// Guarded Ventilation V2 enable
IF L_Vent_V2_Switch_Enabled THEN
    IF NOT L_Vent_V2_Shadow_Diff_Found THEN
        L_Vent_V2_Path_Ready := TRUE;
        L_Vent_Using_Legacy_Fallback := FALSE;
    ELSE
        L_Vent_V2_Path_Ready := FALSE;
        L_Vent_Using_Legacy_Fallback := TRUE;
    END_IF;
ELSE
    L_Vent_V2_Path_Ready := FALSE;
    L_Vent_Using_Legacy_Fallback := TRUE;
END_IF;

// 4. Формирование статусного сообщения
IF L_Policy_Safe_Stop THEN
    VO_Status_Msg := 'ВЕНТИЛЯЦИЯ: ОСТАНОВЛЕНА POLICY SAFE_STOP';
ELSIF L_Policy_Freeze_Protection THEN
    VO_Status_Msg := 'ВЕНТИЛЯЦИЯ: FREEZE_PROTECTION POLICY (stop)';
ELSIF L_Policy_Degraded THEN
    VO_Status_Msg := 'ВЕНТИЛЯЦИЯ: DEGRADED POLICY';
ELSE
    VO_Status_Msg := 'Вентиляция работает в штатном режиме';
END_IF;
// >>> BULK_SYNC_ANCHOR: FB_Ventilation_System_Manager <<<
          
END_FUNCTION_BLOCK

FUNCTION_BLOCK FB_Calibration_Manager
  VAR_INPUT
    VI_Raw_Value : REAL;
    VI_Type : BYTE;
    VI_Calib_Record : ST_Sensor_Calibration_Record;
    VI_System_Time_MS : UDINT;
    VI_Start_Verification : BOOL;
  END_VAR
  VAR_OUTPUT
    VO_Calibrated_Value : REAL;
    VO_Verification_Active : BOOL;
    VO_Verification_Failed : BOOL;
    VO_Deviation_Percent : REAL;
  END_VAR
  VAR
    L_Verification_Timer : FB_System_Timer;
    L_Initial_Value : REAL;
  END_VAR

            // 1. Расчет калиброванного значения
CASE VI_Type OF
    1: VO_Calibrated_Value := VI_Raw_Value + VI_Calib_Record.offset;
    2, 3: VO_Calibrated_Value := (VI_Raw_Value * VI_Calib_Record.multiplier) + VI_Calib_Record.offset;
END_CASE;

// 2. Верификация через 1 час (ТЗ 9.5)
IF VI_Start_Verification AND NOT VO_Verification_Active THEN
    VO_Verification_Active := TRUE;
    L_Initial_Value := VO_Calibrated_Value;
END_IF;

L_Verification_Timer(IN := VO_Verification_Active, PT := T#1h, VI_System_Time_MS := VI_System_Time_MS);

IF L_Verification_Timer.Q THEN
    VO_Verification_Active := FALSE;
    
    // ТЗ 9.5: Отклонение ≤2.0% (норма) / >5.0% (ошибка)
    IF L_Initial_Value <> 0 THEN
        VO_Deviation_Percent := ABS(VO_Calibrated_Value - L_Initial_Value) / L_Initial_Value * 100.0;
    ELSE
        VO_Deviation_Percent := 0.0;
    END_IF;
    
    VO_Verification_Failed := (VO_Deviation_Percent > 5.0);
END_IF;
          
END_FUNCTION_BLOCK

FUNCTION_BLOCK FB_FloorHeating_Controller
  VAR_INPUT
    VI_Current_Temp : REAL;
    VI_Config : ST_FloorHeating_Circuit_Config;
    VI_Tariff : ST_Tariff_Config;
    VI_Current_Hour : UINT;
    VI_IsActivePLC : BOOL;
    VI_System_Time_MS : UDINT;
  END_VAR
  VAR_OUTPUT
    VO_Pump_Run : BOOL;
    VO_Valve_Pos : REAL;
    VO_Valve_Bool : BOOL;
    VO_Effective_Setpoint : REAL;
  END_VAR
  VAR
    L_Is_Night : BOOL;
    L_PID : FB_PID_Controller;
    L_Last_Time : UDINT;
    L_Cycle_Time_S : REAL;
    L_PWM_Period_MS : UDINT;
    L_PWM_Duty_MS : UDINT;
    L_Current_Phase_MS : UDINT;
    L_PWM_Start_Time : UDINT;
  END_VAR

            // Вычисление времени цикла
IF L_Last_Time = 0 THEN
    L_Last_Time := VI_System_Time_MS;
    L_Cycle_Time_S := 1.0;
ELSE
    L_Cycle_Time_S := UDINT_TO_REAL((SEL(VI_System_Time_MS >= L_Last_Time, VI_System_Time_MS - L_Last_Time, (4294967295 - L_Last_Time) + VI_System_Time_MS + 1))) / 1000.0;
    L_Last_Time := VI_System_Time_MS;
END_IF;
IF L_Cycle_Time_S <= 0.0 THEN L_Cycle_Time_S := 0.01; END_IF;

// 1. Определение активного тарифа
IF VI_Tariff.Enabled THEN
    IF VI_Tariff.Night_Start_Hour > VI_Tariff.Night_End_Hour THEN
        // Переход через полночь (например, 23:00 - 07:00)
        L_Is_Night := (VI_Current_Hour >= VI_Tariff.Night_Start_Hour) OR (VI_Current_Hour < VI_Tariff.Night_End_Hour);
    ELSE
        // В пределах одного дня
        L_Is_Night := (VI_Current_Hour >= VI_Tariff.Night_Start_Hour) AND (VI_Current_Hour < VI_Tariff.Night_End_Hour);
    END_IF;
ELSE
    L_Is_Night := FALSE;
END_IF;

// 2. Расчет эффективной уставки
VO_Effective_Setpoint := VI_Config.design_temp;
IF L_Is_Night THEN
    VO_Effective_Setpoint := VO_Effective_Setpoint + VI_Tariff.Boost_Delta;
END_IF;

// 3. ПИД-регулирование
L_PID(
    VI_SetPoint := VO_Effective_Setpoint,
    VI_ProcessValue := VI_Current_Temp,
    VI_Kp := VI_Config.pid_kp,
    VI_Tn := 300.0,
    VI_Tv := 0.0,
    VI_Y_Min := 0.0,
    VI_Y_Max := 100.0,
    VI_Cycle_Time_S := L_Cycle_Time_S,
    VO_Output => VO_Valve_Pos
);

// 4. ШИМ-модуляция для термоэлектрического привода
IF VI_Config.pwm_period_s > 0 THEN
    L_PWM_Period_MS := TO_UDINT(VI_Config.pwm_period_s) * 1000;
ELSE
    L_PWM_Period_MS := 600000; // 10 минут
END_IF;

L_Current_Phase_MS := (SEL(VI_System_Time_MS >= L_PWM_Start_Time, VI_System_Time_MS - L_PWM_Start_Time, (4294967295 - L_PWM_Start_Time) + VI_System_Time_MS + 1));
IF L_Current_Phase_MS >= L_PWM_Period_MS THEN
    L_PWM_Start_Time := VI_System_Time_MS - (L_Current_Phase_MS - L_PWM_Period_MS); // Сохраняем остаток для точности
    L_Current_Phase_MS := (SEL(VI_System_Time_MS >= L_PWM_Start_Time, VI_System_Time_MS - L_PWM_Start_Time, (4294967295 - L_PWM_Start_Time) + VI_System_Time_MS + 1));
END_IF;

L_PWM_Duty_MS := TO_UDINT((VO_Valve_Pos / 100.0) * TO_REAL(L_PWM_Period_MS));

IF VI_IsActivePLC THEN
    VO_Pump_Run := (VO_Valve_Pos > 5.0);
    
    IF VO_Valve_Pos >= 100.0 THEN
        VO_Valve_Bool := TRUE;
    ELSIF VO_Valve_Pos <= 0.0 THEN
        VO_Valve_Bool := FALSE;
    ELSE
        VO_Valve_Bool := (L_Current_Phase_MS <= L_PWM_Duty_MS);
    END_IF;
ELSE
    VO_Pump_Run := FALSE;
    VO_Valve_Bool := FALSE;
END_IF;
          
END_FUNCTION_BLOCK

FUNCTION_BLOCK FB_Fault_Logger
  VAR_INPUT
    VI_Severity : E_System_Severity;
    VI_RootCause : E_System_Root_Cause;
    VI_Time_MS : UDINT;
  END_VAR
  VAR_OUTPUT
    VO_Last_Event_Text : STRING(200);
    VO_Event_Count : UINT;
    VO_Last_Index : UINT;
    VO_Event_Time_MS : ARRAY[1..16] OF UDINT;
    VO_Event_Severity : ARRAY[1..16] OF E_System_Severity;
    VO_Event_RootCause : ARRAY[1..16] OF E_System_Root_Cause;
    VO_Event_Text : ARRAY[1..16] OF STRING(200);
  END_VAR
  VAR
    L_Last_Severity : E_System_Severity;
    L_Last_RootCause : E_System_Root_Cause;
    L_Write_Index : UINT := 0;
    L_Event_Text : STRING(200);
  END_VAR

            L_Event_Text := '';

IF (VI_Severity <> L_Last_Severity) OR (VI_RootCause <> L_Last_RootCause) THEN
    CASE VI_RootCause OF
        E_System_Root_Cause.ROOT_FIRE:
            L_Event_Text := 'EVENT: FIRE DETECTED';
        E_System_Root_Cause.ROOT_GAS_LEAK:
            L_Event_Text := 'EVENT: GAS LEAK';
        E_System_Root_Cause.ROOT_CO_CRITICAL:
            L_Event_Text := 'EVENT: CO CRITICAL';
        E_System_Root_Cause.ROOT_CO_WARNING:
            L_Event_Text := 'EVENT: CO WARNING';
        E_System_Root_Cause.ROOT_WATER_LEAK:
            L_Event_Text := 'EVENT: WATER LEAK';
        E_System_Root_Cause.ROOT_SENSOR_FAULT:
            L_Event_Text := 'EVENT: SENSOR FAULT';
        E_System_Root_Cause.ROOT_IO_OFFLINE:
            L_Event_Text := 'EVENT: IO OFFLINE';
        E_System_Root_Cause.ROOT_COMM_FAULT:
            L_Event_Text := 'EVENT: COMM FAULT';
        E_System_Root_Cause.ROOT_WATCHDOG_FAULT:
            L_Event_Text := 'EVENT: WATCHDOG FAULT';
        E_System_Root_Cause.ROOT_SUBSYSTEM_FAULT:
            L_Event_Text := 'EVENT: SUBSYSTEM FAULT';
        ELSE
            L_Event_Text := 'EVENT: SYSTEM STATE CHANGE';
    END_CASE;

    L_Write_Index := L_Write_Index + 1;
    IF L_Write_Index > 16 THEN
        L_Write_Index := 1;
    END_IF;

    VO_Event_Time_MS[L_Write_Index] := VI_Time_MS;
    VO_Event_Severity[L_Write_Index] := VI_Severity;
    VO_Event_RootCause[L_Write_Index] := VI_RootCause;
    VO_Event_Text[L_Write_Index] := L_Event_Text;

    VO_Last_Index := L_Write_Index;
    VO_Last_Event_Text := L_Event_Text;

    IF VO_Event_Count < 16 THEN
        VO_Event_Count := VO_Event_Count + 1;
    END_IF;
END_IF;

L_Last_Severity := VI_Severity;
L_Last_RootCause := VI_RootCause;
// >>> BULK_SYNC_ANCHOR: FB_Fault_Logger <<<
          
END_FUNCTION_BLOCK

FUNCTION_BLOCK FB_History_Manager
  VAR_INPUT
    VI_System_Time_MS : UDINT;
    VI_Write_Event : BOOL;
    VI_Event : ST_History_Record;
  END_VAR
  VAR_OUTPUT
    VO_Total_Events : UDINT;
  END_VAR
  VAR
    L_Prev_Write_Event : BOOL;
  END_VAR

            IF VI_Write_Event AND NOT L_Prev_Write_Event THEN
    GVL_Retain.G_History_Buffer[GVL_Retain.G_History_Write_Idx] := VI_Event;
    GVL_Retain.G_History_Buffer[GVL_Retain.G_History_Write_Idx].timestamp_ms := VI_System_Time_MS;
    
    GVL_Retain.G_History_Write_Idx := (GVL_Retain.G_History_Write_Idx MOD GVL_CONSTANTS.C_MAX_HISTORY_RECORDS) + 1;
    GVL_Retain.G_History_Total_Events := GVL_Retain.G_History_Total_Events + 1;
END_IF;
L_Prev_Write_Event := VI_Write_Event;

VO_Total_Events := GVL_Retain.G_History_Total_Events;
// >>> BULK_SYNC_ANCHOR: FB_History_Manager <<<
          
END_FUNCTION_BLOCK

FUNCTION_BLOCK FB_Watchdog
  VAR_INPUT
    VI_System_Time_MS : UDINT;
    VI_Timeout_MS : UDINT := 2000;
  END_VAR
  VAR_OUTPUT
    VO_Alive : BOOL;
    VO_Watchdog_Fault : BOOL;
    VO_Cycle_DT_MS : UDINT;
  END_VAR
  VAR
    L_Initialized : BOOL := FALSE;
    L_Last_Call_MS : UDINT := 0;
    L_DT_MS : UDINT := 0;
  END_VAR

            IF NOT L_Initialized THEN
    L_Initialized := TRUE;
    L_Last_Call_MS := VI_System_Time_MS;
    VO_Cycle_DT_MS := 0;
    VO_Watchdog_Fault := FALSE;
    VO_Alive := TRUE;
    RETURN;
END_IF;

// Measure real time gap between successive calls
L_DT_MS := (SEL(VI_System_Time_MS >= L_Last_Call_MS, VI_System_Time_MS - L_Last_Call_MS, (4294967295 - L_Last_Call_MS) + VI_System_Time_MS + 1));
VO_Cycle_DT_MS := L_DT_MS;

// Fault if the task/cycle resumed after an abnormal pause
VO_Watchdog_Fault := (L_DT_MS > VI_Timeout_MS);
VO_Alive := NOT VO_Watchdog_Fault;

// Store current timestamp for next cycle
L_Last_Call_MS := VI_System_Time_MS;
// >>> BULK_SYNC_ANCHOR: FB_Watchdog <<<
          
END_FUNCTION_BLOCK

FUNCTION_BLOCK FB_Blinds_V2_Staging
  VAR_INPUT
    VI_Blind_ID : INT;
    VI_Enable : BOOL;
    VI_Position_Setpoint : BYTE;
    VI_Manual_Override : BOOL;
    VI_Scenario_ID : INT;
    VI_Safety_Mode : BOOL;
    VI_Position_Actual : BYTE;
    VI_Manual_Override_Active : BOOL;
    VI_Is_Moving : BOOL;
    VI_Alarm_Active : BOOL;
  END_VAR
  VAR_OUTPUT
    VO_Command_Shadow : ST_Blinds_Command_V2;
    VO_State_Shadow : ST_Blinds_State_V2;
  END_VAR

            VO_Command_Shadow.Position_Setpoint := VI_Position_Setpoint;
VO_State_Shadow.Position_Actual := VI_Position_Actual;
          
END_FUNCTION_BLOCK

FUNCTION_BLOCK FB_IO_Module_Watchdog
  VAR_INPUT
    VI_System_Time_MS : UDINT;
    VI_Module_ID : BYTE;
    VI_Heartbeat_Signal : BOOL;
    VI_Timeout_MS : UDINT := 2000;
  END_VAR
  VAR_OUTPUT
    VO_Module_Online : BOOL;
    VO_Error_Active : BOOL;
  END_VAR
  VAR
    L_Last_Heartbeat_State : BOOL;
    L_Last_Heartbeat_Time : UDINT;
    L_Elapsed_Time : UDINT;
  END_VAR

            // Отслеживание изменения сигнала
IF VI_Heartbeat_Signal <> L_Last_Heartbeat_State THEN
    L_Last_Heartbeat_Time := VI_System_Time_MS;
    L_Last_Heartbeat_State := VI_Heartbeat_Signal;
END_IF;

// Проверка таймаута
L_Elapsed_Time := (SEL(VI_System_Time_MS >= L_Last_Heartbeat_Time, VI_System_Time_MS - L_Last_Heartbeat_Time, (4294967295 - L_Last_Heartbeat_Time) + VI_System_Time_MS + 1));

IF L_Elapsed_Time > VI_Timeout_MS THEN
    VO_Module_Online := FALSE;
    VO_Error_Active := TRUE;
ELSE
    VO_Module_Online := TRUE;
    VO_Error_Active := FALSE;
END_IF;
// >>> BULK_SYNC_ANCHOR: FB_IO_Module_Watchdog <<<
          
END_FUNCTION_BLOCK

FUNCTION_BLOCK FB_AccessCode_Manager
  VAR_INPUT
    VI_System_Time_MS : UDINT;
    VI_IsActivePLC : BOOL;
    VI_Code_To_Check : STRING(4);
    VI_RFID_To_Check : STRING(20);
  END_VAR
  VAR_OUTPUT
    VO_Code_Valid : BOOL;
  END_VAR
  VAR_IN_OUT
    VI_Access_Codes : ARRAY[1..GVL_CONSTANTS.C_MAX_ACCESS_CODES] OF DWORD;
    VI_RFID_Tags : ARRAY[1..GVL_CONSTANTS.C_MAX_ACCESS_CODES] OF STRING(20);
  END_VAR
  VAR
    L_i : INT;
    pCode : POINTER TO BYTE;
    L_CRC_Calc : FB_CRC32_Calculator;
    L_Input_Hash : DWORD;
  END_VAR

            VO_Code_Valid := FALSE;

// Вычисляем хэш введенного кода
IF LEN(VI_Code_To_Check) > 0 THEN
    pCode := ADR(VI_Code_To_Check);
    L_Input_Hash := 0;
    FOR L_i := 1 TO GVL_CONSTANTS.C_MAX_ACCESS_CODES DO
        IF VI_Access_Codes[L_i] <> 0 AND VI_Access_Codes[L_i] = L_Input_Hash THEN
            VO_Code_Valid := TRUE;
            RETURN;
        END_IF;
    END_FOR;
END_IF;

// Проверяем RFID метку
IF LEN(VI_RFID_To_Check) > 0 THEN
    FOR L_i := 1 TO GVL_CONSTANTS.C_MAX_ACCESS_CODES DO
        IF VI_RFID_Tags[L_i] <> '' AND VI_RFID_Tags[L_i] = VI_RFID_To_Check THEN
            VO_Code_Valid := TRUE;
            RETURN;
        END_IF;
    END_FOR;
END_IF;
// >>> BULK_SYNC_ANCHOR: FB_AccessCode_Manager <<<
          
END_FUNCTION_BLOCK

FUNCTION_BLOCK FB_State_Snapshot_Manager
  VAR_INPUT
    VI_System_Time_MS : UDINT;
    VI_Trigger_Event : BOOL;
    VI_Event_Code : WORD;
    VI_Current_State : ST_State_Snapshot;
  END_VAR
  VAR_OUTPUT
    VO_Snapshot_Saved : BOOL;
  END_VAR
  VAR
    L_Snapshot_Buffer : ARRAY[1..GVL_CONSTANTS.C_MAX_STATE_SNAPSHOTS] OF ST_State_Snapshot;
    L_Write_Idx : INT := 1;
  END_VAR

            IF VI_Trigger_Event THEN
    L_Snapshot_Buffer[L_Write_Idx] := VI_Current_State;
    L_Snapshot_Buffer[L_Write_Idx].timestamp_ms := VI_System_Time_MS;
    L_Snapshot_Buffer[L_Write_Idx].trigger_event_code := VI_Event_Code;
    
    L_Write_Idx := (L_Write_Idx MOD GVL_CONSTANTS.C_MAX_STATE_SNAPSHOTS) + 1;
    VO_Snapshot_Saved := TRUE;
ELSE
    VO_Snapshot_Saved := FALSE;
END_IF;
          
END_FUNCTION_BLOCK

FUNCTION_BLOCK FB_Trend_Analyzer
  VAR_INPUT
    VI_Count : INT;
  END_VAR
  VAR_OUTPUT
    VO_Average : REAL;
    VO_Max : REAL;
    VO_Min : REAL;
    VO_Trend_Up : BOOL;
    VO_Trend_Down : BOOL;
  END_VAR
  VAR_IN_OUT
    VI_Data : ARRAY[1..GVL_CONSTANTS.C_MAX_TREND_DATA_POINTS] OF REAL;
  END_VAR
  VAR
    L_i : INT;
    L_Sum : REAL;
  END_VAR

            IF VI_Count > 0 AND VI_Count <= GVL_CONSTANTS.C_MAX_TREND_DATA_POINTS THEN
    VO_Max := VI_Data[1];
    VO_Min := VI_Data[1];
    L_Sum := 0.0;
    
    FOR L_i := 1 TO VI_Count DO
        IF VI_Data[L_i] > VO_Max THEN VO_Max := VI_Data[L_i]; END_IF;
        IF VI_Data[L_i] < VO_Min THEN VO_Min := VI_Data[L_i]; END_IF;
        L_Sum := L_Sum + VI_Data[L_i];
    END_FOR;
    
    VO_Average := L_Sum / INT_TO_REAL(VI_Count);
    
    IF VI_Count >= 2 THEN
        VO_Trend_Up := (VI_Data[VI_Count] > VI_Data[1]);
        VO_Trend_Down := (VI_Data[VI_Count] < VI_Data[1]);
    END_IF;
END_IF;
          
END_FUNCTION_BLOCK

FUNCTION_BLOCK FB_System_Timer_TOF
  VAR_INPUT
    IN : BOOL;
    PT : TIME;
    VI_System_Time_MS : UDINT;
  END_VAR
  VAR_OUTPUT
    Q : BOOL;
    ET : TIME;
  END_VAR
  VAR
    L_Start_Time : UDINT;
    L_Running : BOOL;
    L_Prev_IN : BOOL;
  END_VAR

            // ==============================================================================
// Блок таймера задержки выключения (System Timer TOF)
// Назначение:
// - Замена стандартного TOF для обеспечения точной выдержки времени,
//   независимой от времени цикла ПЛК, с использованием единого системного времени.
// ==============================================================================



IF IN THEN
    Q := TRUE;
    ET := T#0s;
    L_Running := FALSE;
ELSE
    IF L_Prev_IN THEN
        L_Start_Time := VI_System_Time_MS;
        L_Running := TRUE;
        ET := T#0s;
    END_IF;
    
    IF L_Running THEN
        // Обработка переполнения UDINT (примерно 49 дней)
        ET := TO_TIME((SEL(VI_System_Time_MS >= L_Start_Time, VI_System_Time_MS - L_Start_Time, (4294967295 - L_Start_Time) + VI_System_Time_MS + 1)));
        
        IF ET >= PT THEN
            Q := FALSE;
            ET := PT;
            L_Running := FALSE;
        ELSE
            Q := TRUE;
        END_IF;
    END_IF;
END_IF;

L_Prev_IN := IN;
          
END_FUNCTION_BLOCK

FUNCTION_BLOCK FB_State_Replication
  VAR_INPUT
    VI_Local_Role : E_PLC_ROLE;
    VI_Sync_Req : BOOL;
    VI_Local_State : ST_System_State_Snapshot;
    VI_Remote_State : ST_System_State_Snapshot;
    VI_System_Time_MS : UDINT;
  END_VAR
  VAR_OUTPUT
    VO_State_Updated : BOOL;
    VO_Synced_State : ST_System_State_Snapshot;
  END_VAR
  VAR
    L_Sync_In_Progress : BOOL;
    L_Last_Sync_Time : UDINT;
    L_Periodic_Sync_Req : BOOL;
    L_Elapsed_Time : UDINT;
  END_VAR

            // Периодическая синхронизация (каждые 5 секунд)
L_Elapsed_Time := (SEL(VI_System_Time_MS >= L_Last_Sync_Time, VI_System_Time_MS - L_Last_Sync_Time, (4294967295 - L_Last_Sync_Time) + VI_System_Time_MS + 1));

IF L_Elapsed_Time > 5000 THEN
    L_Periodic_Sync_Req := TRUE;
    L_Last_Sync_Time := VI_System_Time_MS;
ELSE
    L_Periodic_Sync_Req := FALSE;
END_IF;

// State Replication Logic
// Синхронизация состояния между ПЛК (ТЗ 8.2)
IF (VI_Sync_Req OR L_Periodic_Sync_Req) AND NOT L_Sync_In_Progress THEN
    L_Sync_In_Progress := TRUE;
    
    // Разрешение конфликтов на основе версии состояния
    IF VI_Remote_State.Version > VI_Local_State.Version THEN
        VO_Synced_State := VI_Remote_State;
        VO_State_Updated := TRUE;
    ELSIF VI_Remote_State.Version = VI_Local_State.Version THEN
        // Если версии равны, приоритет у ведущего ПЛК
        IF VI_Local_Role = E_PLC_ROLE.ROLE_STANDBY THEN
            VO_Synced_State := VI_Remote_State;
            VO_State_Updated := TRUE;
        ELSE
            VO_Synced_State := VI_Local_State;
            VO_State_Updated := FALSE;
        END_IF;
    ELSE
        VO_Synced_State := VI_Local_State;
        VO_State_Updated := FALSE;
    END_IF;
ELSIF NOT (VI_Sync_Req OR L_Periodic_Sync_Req) THEN
    L_Sync_In_Progress := FALSE;
    VO_State_Updated := FALSE;
    VO_Synced_State := VI_Local_State;
END_IF;
          
END_FUNCTION_BLOCK

FUNCTION_BLOCK FB_Boiler_OpenTherm_Interface
  VAR_INPUT
    VI_Enable : ARRAY[1..GVL_CONSTANTS.C_MAX_BOILERS] OF BOOL;
    VI_Setpoint : ARRAY[1..GVL_CONSTANTS.C_MAX_BOILERS] OF REAL;
    VI_OT_Online : ARRAY[1..GVL_CONSTANTS.C_MAX_BOILERS] OF BOOL;
    VI_OT_Error : ARRAY[1..GVL_CONSTANTS.C_MAX_BOILERS] OF BOOL;
  END_VAR
  VAR_OUTPUT
    VO_OT_Enable : ARRAY[1..GVL_CONSTANTS.C_MAX_BOILERS] OF BOOL;
    VO_OT_Setpoint : ARRAY[1..GVL_CONSTANTS.C_MAX_BOILERS] OF REAL;
    VO_OT_Command_Valid : ARRAY[1..GVL_CONSTANTS.C_MAX_BOILERS] OF BOOL;
  END_VAR
  VAR
    L_i : INT;
  END_VAR

            FOR L_i := 1 TO GVL_CONSTANTS.C_MAX_BOILERS DO
    VO_OT_Enable[L_i] := FALSE;
    VO_OT_Setpoint[L_i] := 0.0;
    VO_OT_Command_Valid[L_i] := FALSE;

    IF VI_Enable[L_i] AND VI_OT_Online[L_i] AND NOT VI_OT_Error[L_i] THEN
        VO_OT_Enable[L_i] := TRUE;
        VO_OT_Setpoint[L_i] := LIMIT(20.0, VI_Setpoint[L_i], 80.0);
        VO_OT_Command_Valid[L_i] := TRUE;
    END_IF;
END_FOR;
          
END_FUNCTION_BLOCK

FUNCTION_BLOCK FB_FloorHeating_Overheat_Protection
  VAR_INPUT
    VI_Threshold : REAL := 45.0;
  END_VAR
  VAR_OUTPUT
    VO_Overheat_Detected : BOOL;
    VO_Locked_Circuits : ARRAY[1..GVL_CONSTANTS.C_MAX_HEATING_CIRCUITS] OF BOOL;
  END_VAR
  VAR_IN_OUT
    VI_Temps : ARRAY[1..GVL_CONSTANTS.C_MAX_HEATING_CIRCUITS] OF REAL;
  END_VAR
  VAR
    L_i : INT;
  END_VAR

            VO_Overheat_Detected := FALSE;
FOR L_i := 1 TO GVL_CONSTANTS.C_MAX_HEATING_CIRCUITS DO
    IF VI_Temps[L_i] > VI_Threshold THEN
        VO_Overheat_Detected := TRUE;
        VO_Locked_Circuits[L_i] := TRUE;
    END_IF;
END_FOR;
          
END_FUNCTION_BLOCK

FUNCTION_BLOCK FB_Pre_Departure_Heating
  VAR_INPUT
    VI_Departure_Time : UDINT;
    VI_System_Time : UDINT;
  END_VAR
  VAR_OUTPUT
    VO_Heating_Active : BOOL;
    VO_Setpoints : ARRAY[1..GVL_CONSTANTS.C_MAX_HEATING_CIRCUITS] OF REAL;
  END_VAR
  VAR_IN_OUT
    VI_Selected : ARRAY[1..GVL_CONSTANTS.C_MAX_HEATING_CIRCUITS] OF BOOL;
  END_VAR
  VAR
    L_i : INT;
  END_VAR

            // Запуск за 3 часа (10800000 мс)
IF (SEL(VI_Departure_Time >= VI_System_Time, VI_Departure_Time - VI_System_Time, (4294967295 - VI_System_Time) + VI_Departure_Time + 1)) < 10800000 THEN
    VO_Heating_Active := TRUE;
    FOR L_i := 1 TO GVL_CONSTANTS.C_MAX_HEATING_CIRCUITS DO
        IF VI_Selected[L_i] THEN VO_Setpoints[L_i] := 22.0; END_IF;
    END_FOR;
ELSE
    VO_Heating_Active := FALSE;
END_IF;
          
END_FUNCTION_BLOCK

FUNCTION_BLOCK FB_PID_Controller
  VAR_INPUT
    VI_SetPoint : REAL;
    VI_ProcessValue : REAL;
    VI_Kp : REAL;
    VI_Tn : REAL;
    VI_Tv : REAL;
    VI_Y_Min : REAL := 0.0;
    VI_Y_Max : REAL := 100.0;
    VI_Manual_Mode : BOOL;
    VI_Manual_Value : REAL;
    VI_Deadband : REAL := 0.1;
    VI_Cycle_Time_S : REAL := 0.01;
    VI_Reset : BOOL;
  END_VAR
  VAR_OUTPUT
    VO_Output : REAL;
    VO_Error : REAL;
    VO_Limiting : BOOL;
  END_VAR
  VAR
    L_Integral_Sum : REAL;
    L_Prev_Error : REAL;
    L_Derivative : REAL;
    L_Output_Raw : REAL;
  END_VAR

            // Расчет ошибки
VO_Error := VI_SetPoint - VI_ProcessValue;

// Проверка мертвой зоны
IF ABS(VO_Error) < VI_Deadband THEN
    VO_Error := 0.0;
END_IF;

IF VI_Reset THEN
    L_Integral_Sum := 0.0;
    L_Prev_Error := 0.0;
    VO_Output := 0.0;
    RETURN;
END_IF;

IF VI_Manual_Mode THEN
    VO_Output := VI_Manual_Value;
    // Безударный переход: при выходе из ручного режима выход должен остаться прежним.
    // Так как Выход = P + I + D, то I = Выход - P - D.
    // Для простоты D при переходе обнуляем (или игнорируем), тогда I = Выход - P.
    L_Integral_Sum := VO_Output - (VI_Kp * VO_Error);
    L_Prev_Error := VO_Error;
    RETURN;
END_IF;

// Пропорциональная составляющая
L_Output_Raw := VI_Kp * VO_Error;

// Интегральная составляющая (Метод трапеций)
IF VI_Tn > 0.0 THEN
    // Anti-windup: не накапливаем интеграл, если выход уже на пределе и ошибка того же знака
    IF NOT VO_Limiting OR (VO_Error > 0.0 AND L_Output_Raw < VI_Y_Max) OR (VO_Error < 0.0 AND L_Output_Raw > VI_Y_Min) THEN
        L_Integral_Sum := L_Integral_Sum + (VI_Kp / VI_Tn) * VO_Error * VI_Cycle_Time_S;
    END_IF;
    L_Output_Raw := L_Output_Raw + L_Integral_Sum;
END_IF;

// Дифференциальная составляющая
IF VI_Tv > 0.0 THEN
    L_Derivative := (VO_Error - L_Prev_Error) / VI_Cycle_Time_S;
    L_Output_Raw := L_Output_Raw + VI_Kp * VI_Tv * L_Derivative;
END_IF;

L_Prev_Error := VO_Error;

// Ограничение выхода
IF L_Output_Raw > VI_Y_Max THEN
    VO_Output := VI_Y_Max;
    VO_Limiting := TRUE;
ELSIF L_Output_Raw < VI_Y_Min THEN
    VO_Output := VI_Y_Min;
    VO_Limiting := TRUE;
ELSE
    VO_Output := L_Output_Raw;
    VO_Limiting := FALSE;
END_IF;
// >>> BULK_SYNC_ANCHOR: FB_PID_Controller <<<
          
END_FUNCTION_BLOCK

FUNCTION_BLOCK FB_SHA1
  VAR_INPUT
    Length : INT;
  END_VAR
  VAR_OUTPUT
    Hash : ARRAY[0..19] OF BYTE;
  END_VAR
  VAR_IN_OUT
    Data : ARRAY[0..127] OF BYTE;
  END_VAR
  VAR
    H0, H1, H2, H3, H4 : DWORD;
    A, B, C, D, E, F, K, Temp : DWORD;
    W : ARRAY[0..79] OF DWORD;
    i, j, t : INT;
    PaddedData : ARRAY[0..127] OF BYTE;
    PaddedLength : INT;
    NumBlocks : INT;
    BlockOffset : INT;
  END_VAR

            // Initialize variables
H0 := 16#67452301;
H1 := 16#EFCDAB89;
H2 := 16#98BADCFE;
H3 := 16#10325476;
H4 := 16#C3D2E1F0;

// Pre-processing
FOR i := 0 TO Length - 1 DO
    PaddedData[i] := Data[i];
END_FOR;

// Append the bit '1' to the message
PaddedData[Length] := 16#80;

// Append 0 <= k < 512 bits '0', such that the resulting message length in bits
// is congruent to -64 ≡ 448 (mod 512)
PaddedLength := Length + 1;
WHILE (PaddedLength MOD 64) <> 56 DO
    PaddedData[PaddedLength] := 0;
    PaddedLength := PaddedLength + 1;
END_WHILE;

// Append length of message (before pre-processing), in bits, as 64-bit big-endian integer
// Since our message is small (max 127 bytes), we only need the lower 32 bits
Temp := TO_DWORD(Length * 8);
PaddedData[PaddedLength] := 0;
PaddedData[PaddedLength+1] := 0;
PaddedData[PaddedLength+2] := 0;
PaddedData[PaddedLength+3] := 0;
PaddedData[PaddedLength+4] := TO_BYTE(SHR(Temp, 24));
PaddedData[PaddedLength+5] := TO_BYTE(SHR(Temp, 16));
PaddedData[PaddedLength+6] := TO_BYTE(SHR(Temp, 8));
PaddedData[PaddedLength+7] := TO_BYTE(Temp);
PaddedLength := PaddedLength + 8;

NumBlocks := PaddedLength / 64;

// Process the message in successive 512-bit chunks
FOR i := 0 TO NumBlocks - 1 DO
    BlockOffset := i * 64;
    
    // Break chunk into sixteen 32-bit big-endian words w[i], 0 <= i <= 15
    FOR j := 0 TO 15 DO
        W[j] := SHL(TO_DWORD(PaddedData[BlockOffset + j*4]), 24) OR
                SHL(TO_DWORD(PaddedData[BlockOffset + j*4 + 1]), 16) OR
                SHL(TO_DWORD(PaddedData[BlockOffset + j*4 + 2]), 8) OR
                TO_DWORD(PaddedData[BlockOffset + j*4 + 3]);
    END_FOR;
    
    // Message schedule: extend the sixteen 32-bit words into eighty 32-bit words
    FOR j := 16 TO 79 DO
        Temp := W[j-3] XOR W[j-8] XOR W[j-14] XOR W[j-16];
        W[j] := SHL(Temp, 1) OR SHR(Temp, 31); // Left rotate by 1
    END_FOR;
    
    // Initialize hash value for this chunk
    A := H0;
    B := H1;
    C := H2;
    D := H3;
    E := H4;
    
    // Main loop
    FOR j := 0 TO 79 DO
        IF j <= 19 THEN
            F := (B AND C) OR ((NOT B) AND D);
            K := 16#5A827999;
        ELSIF j <= 39 THEN
            F := B XOR C XOR D;
            K := 16#6ED9EBA1;
        ELSIF j <= 59 THEN
            F := (B AND C) OR (B AND D) OR (C AND D);
            K := 16#8F1BBCDC;
        ELSE
            F := B XOR C XOR D;
            K := 16#CA62C1D6;
        END_IF;
        
        Temp := (SHL(A, 5) OR SHR(A, 27)) + F + E + K + W[j];
        E := D;
        D := C;
        C := SHL(B, 30) OR SHR(B, 2);
        B := A;
        A := Temp;
    END_FOR;
    
    // Add this chunk's hash to result so far
    H0 := H0 + A;
    H1 := H1 + B;
    H2 := H2 + C;
    H3 := H3 + D;
    H4 := H4 + E;
END_FOR;

// Produce the final hash value (big-endian)
Hash[0] := TO_BYTE(SHR(H0, 24)); Hash[1] := TO_BYTE(SHR(H0, 16)); Hash[2] := TO_BYTE(SHR(H0, 8)); Hash[3] := TO_BYTE(H0);
Hash[4] := TO_BYTE(SHR(H1, 24)); Hash[5] := TO_BYTE(SHR(H1, 16)); Hash[6] := TO_BYTE(SHR(H1, 8)); Hash[7] := TO_BYTE(H1);
Hash[8] := TO_BYTE(SHR(H2, 24)); Hash[9] := TO_BYTE(SHR(H2, 16)); Hash[10] := TO_BYTE(SHR(H2, 8)); Hash[11] := TO_BYTE(H2);
Hash[12] := TO_BYTE(SHR(H3, 24)); Hash[13] := TO_BYTE(SHR(H3, 16)); Hash[14] := TO_BYTE(SHR(H3, 8)); Hash[15] := TO_BYTE(H3);
Hash[16] := TO_BYTE(SHR(H4, 24)); Hash[17] := TO_BYTE(SHR(H4, 16)); Hash[18] := TO_BYTE(SHR(H4, 8)); Hash[19] := TO_BYTE(H4);
          
END_FUNCTION_BLOCK

FUNCTION_BLOCK FB_Sensor_Distribution
  VAR_INPUT
    VI_Raw_Temp : REAL;
    VI_Raw_Hum : REAL;
    VI_Raw_CO2 : REAL;
  END_VAR
  VAR_OUTPUT
    VO_Temp_Heating : REAL;
    VO_Temp_Vent : REAL;
    VO_Hum_Vent : REAL;
    VO_CO2_Vent : REAL;
  END_VAR

            // Распределение данных по подсистемам
VO_Temp_Heating := VI_Raw_Temp;
VO_Temp_Vent    := VI_Raw_Temp;
VO_Hum_Vent     := VI_Raw_Hum;
VO_CO2_Vent     := VI_Raw_CO2;
          
END_FUNCTION_BLOCK

FUNCTION_BLOCK FB_BlackBox_V2_Core
  VAR_INPUT
    VI_System_Time_MS : UDINT;
    VI_System_Mode : INT;
    VI_Critical_Alarm_Active : BOOL;
    VI_Warning_Active : BOOL;
    VI_First_Fault_Type : BYTE;
    VI_First_Fault_Source : BYTE;
    VI_Gas_Alarm : BOOL;
    VI_Fire_Alarm : BOOL;
    VI_Flood_Alarm : BOOL;
  END_VAR
  VAR_OUTPUT
    VO_Snapshot : ST_BlackBox_Snapshot_V2;
  END_VAR

            VO_Snapshot.Gas_Alarm := VI_Gas_Alarm;
VO_Snapshot.Fire_Alarm := VI_Fire_Alarm;
VO_Snapshot.Flood_Alarm := VI_Flood_Alarm;
VO_Snapshot.First_Fault_Type := VI_First_Fault_Type;
VO_Snapshot.First_Fault_Source := VI_First_Fault_Source;
          
END_FUNCTION_BLOCK

FUNCTION_BLOCK FB_Presence_Simulator
  VAR_INPUT
    VI_Enabled : BOOL;
    VI_Intensity : REAL;
    VI_System_Time : UDINT;
    VI_Use_Playback : BOOL;
  END_VAR
  VAR_OUTPUT
    VO_Light_States : ARRAY[1..32] OF BOOL;
  END_VAR
  VAR
    fbPlayback : FB_Presence_Playback;
  END_VAR

            IF VI_Enabled THEN
    IF VI_Use_Playback THEN
        fbPlayback(VI_Mode_Record := FALSE, VI_Time_Index := VI_System_Time MOD 604800000, VO_Light_Outputs => VO_Light_States);
    ELSE
        // Старая логика случайной симуляции
        VO_Light_States[1] := (VI_System_Time MOD 100000 > 50000);
    END_IF;
END_IF;
          
END_FUNCTION_BLOCK

FUNCTION_BLOCK FB_Alarm_Compatibility_Package
  VAR_INPUT
    VI_Alarm_Legacy : ST_Alarm_Record;
  END_VAR
  VAR_OUTPUT
    VO_OK : BOOL;
    VO_Alarm_Legacy_Roundtrip : ST_Alarm_Record;
  END_VAR

            VO_OK := TRUE;
VO_Alarm_Legacy_Roundtrip := VI_Alarm_Legacy;
          
END_FUNCTION_BLOCK

FUNCTION_BLOCK FB_Emergency_Valve_Open
  VAR_INPUT
    VI_Fire_Alarm : BOOL;
    VI_Gas_Alarm : BOOL;
  END_VAR
  VAR_OUTPUT
    VO_Open_Cmd : BOOL;
  END_VAR

            // Приоритетное открытие при любой серьезной аварии
VO_Open_Cmd := VI_Fire_Alarm OR VI_Gas_Alarm;
          
END_FUNCTION_BLOCK

FUNCTION_BLOCK FB_Lighting_Blinds_Manager
  VAR_INPUT
    VI_System_Time_MS : UDINT;
    VI_IsActivePLC : BOOL;
    VI_Current_Scenario : E_SCENARIO_TYPE;
    VI_Away_Level : BYTE;
    VI_Simulation_Active : BOOL;
    VI_Is_Night : BOOL;
    VI_System_Mode : E_System_Operating_Mode;
  END_VAR
  VAR_OUTPUT
    VO_Lighting_Levels : ARRAY[1..32] OF BYTE;
    VO_Blinds_Positions : ARRAY[1..GVL_CONSTANTS.C_MAX_BLINDS] OF BYTE;
    VO_Wet_Zone_Light_Active : ARRAY[1..GVL_CONSTANTS.C_MAX_WET_ZONES] OF BOOL;
  END_VAR
  VAR_IN_OUT
    VI_Manual_Light_Override : ARRAY[1..32] OF BYTE;
    VI_Manual_Blinds_Override : ARRAY[1..GVL_CONSTANTS.C_MAX_BLINDS] OF BYTE;
    VI_Simulation_Lights : ARRAY[1..32] OF BOOL;
    VI_Physical_Switches : ARRAY[1..32] OF BOOL;
    VI_Motion_Sensors : ARRAY[1..32] OF BOOL;
    VI_Rule_Actions : ARRAY[1..GVL_CONSTANTS.C_MAX_RULES] OF ST_Rule_Action;
    VI_IO_Modules_Online : ARRAY[1..GVL_CONSTANTS.C_MAX_MODULES] OF BOOL;
    VI_Wet_Zone_Map : ARRAY[1..32] OF BOOL;
    VI_Scenario_Configs : ARRAY[1..GVL_CONSTANTS.C_MAX_SCENARIOS] OF ST_Scenario_Config;
  END_VAR
  VAR
    fbBlindsV2Staging : FB_Blinds_V2_Staging;
    L_Blinds_V2_Command_Shadow : ST_Blinds_Command_V2;
    L_Blinds_V2_State_Shadow : ST_Blinds_State_V2;
    L_Blinds_V2_Shadow_Diff_Found : BOOL;
    L_Blinds_V2_Switch_Enabled : BOOL;
    L_Blinds_V2_Path_Ready : BOOL;
    L_Blinds_Using_Legacy_Fallback : BOOL;
    fbLightingV2Staging : FB_Lighting_V2_Staging;
    L_Lighting_V2_Command_Shadow : ST_Lighting_Command_V2;
    L_Lighting_V2_State_Shadow : ST_Lighting_State_V2;
    L_Lighting_V2_Shadow_Diff_Found : BOOL;
    L_Lighting_V2_Switch_Enabled : BOOL;
    L_Lighting_V2_Path_Ready : BOOL;
    L_Lighting_Using_Legacy_Fallback : BOOL;
    L_i : INT;
    L_j : INT;
    L_Base_Light : BYTE;
    L_Base_Blinds : BYTE;
    L_Target_Base_Light : BYTE;
    L_Target_Base_Blinds : BYTE;
    L_Prev_Scenario : E_SCENARIO_TYPE;
    L_Transition_Light : FB_Scenario_Transition_Controller;
    L_Transition_Blinds : FB_Scenario_Transition_Controller;
    L_Light_States : ARRAY[1..32] OF BOOL;
    L_Prev_Switches : ARRAY[1..32] OF BOOL;
    L_Prev_Motion_Q : ARRAY[1..32] OF BOOL;
    L_Manual_Override : ARRAY[1..32] OF BOOL;
    L_Motion_Timers : ARRAY[1..32] OF FB_System_Timer_TOF;
    L_Rule_Light_Active : BOOL;
    L_Rule_Light_Val : BYTE;
    L_Rule_Blinds_Active : BOOL;
    L_Rule_Blinds_Val : BYTE;
    L_Wet_Zone_Idx : INT;
    L_Effective_Scenario : E_SCENARIO_TYPE;
    L_Effective_Simulation_Active : BOOL;
  END_VAR

            // Менеджер управления освещением и шторами/жалюзи.
// Обеспечивает работу по сценариями, датчикам движения, физическим выключателям и правилам.


IF NOT VI_IsActivePLC THEN RETURN; END_IF;

L_Lighting_V2_Shadow_Diff_Found := FALSE;
L_Blinds_V2_Shadow_Diff_Found := FALSE;
L_Blinds_V2_Switch_Enabled := TRUE;
L_Blinds_V2_Path_Ready := FALSE;
L_Blinds_Using_Legacy_Fallback := TRUE;
L_Lighting_V2_Switch_Enabled := TRUE;
L_Lighting_V2_Path_Ready := FALSE;
L_Lighting_Using_Legacy_Fallback := TRUE;

GVL_STATE.G_Lighting_IO_Fault := FALSE;
GVL_STATE.G_Lighting_Subsystem_Degraded := FALSE;

L_Effective_Scenario := VI_Current_Scenario;
L_Effective_Simulation_Active := VI_Simulation_Active;

CASE VI_System_Mode OF
    E_System_Operating_Mode.MODE_SAFE_STOP:
        FOR L_j := 1 TO 32 DO
            VO_Lighting_Levels[L_j] := 0;
        END_FOR;
        FOR L_j := 1 TO GVL_CONSTANTS.C_MAX_BLINDS DO
            VO_Blinds_Positions[L_j] := 100;
        END_FOR;
        FOR L_j := 1 TO GVL_CONSTANTS.C_MAX_WET_ZONES DO
            VO_Wet_Zone_Light_Active[L_j] := FALSE;
        END_FOR;
        RETURN;
    E_System_Operating_Mode.MODE_FREEZE_PROTECTION:
        L_Effective_Scenario := E_SCENARIO_TYPE.SCENARIO_NONE;
        L_Effective_Simulation_Active := FALSE;
    E_System_Operating_Mode.MODE_DEGRADED:
        L_Effective_Simulation_Active := FALSE;
END_CASE;

// Инициализация индекса мокрых зон
L_Wet_Zone_Idx := 1;
// Сброс массива мокрых зон
FOR L_i := 1 TO GVL_CONSTANTS.C_MAX_WET_ZONES DO
    VO_Wet_Zone_Light_Active[L_i] := FALSE;
END_FOR;

// Проверка связи с модулями ввода-вывода
FOR L_i := 1 TO GVL_CONSTANTS.C_MAX_MODULES DO
    IF NOT VI_IO_Modules_Online[L_i] THEN
        GVL_STATE.G_Lighting_IO_Fault := TRUE;
GVL_STATE.G_Lighting_Subsystem_Degraded := TRUE;
        // Переход в безопасное состояние при потере связи (свет выкл, шторы открыты для эвакуации)
        FOR L_j := 1 TO 32 DO
            VO_Lighting_Levels[L_j] := 0;
        END_FOR;
        FOR L_j := 1 TO GVL_CONSTANTS.C_MAX_BLINDS DO
            VO_Blinds_Positions[L_j] := 100;
        END_FOR;
        RETURN;
    END_IF;
END_FOR;

// 1. Определение целевых уровней по сценарию (ТЗ 7.1)
IF L_Effective_Scenario >= 1 AND L_Effective_Scenario <= GVL_CONSTANTS.C_MAX_SCENARIOS THEN
    L_Target_Base_Light := VI_Scenario_Configs[L_Effective_Scenario].lighting_level_base;
    L_Target_Base_Blinds := VI_Scenario_Configs[L_Effective_Scenario].blinds_position_percent;
ELSE
    L_Target_Base_Light := 100;
    L_Target_Base_Blinds := 100;
END_IF;

// Корректировка по астрономическому таймеру
IF VI_Is_Night AND L_Effective_Scenario <> E_SCENARIO_TYPE.SCENARIO_AWAY AND L_Effective_Scenario <> E_SCENARIO_TYPE.SCENARIO_SLEEP THEN
    L_Target_Base_Blinds := 0; // Закрывать шторы ночью
END_IF;

// Плавный переход при смене сценария
IF L_Effective_Scenario <> L_Prev_Scenario THEN
    L_Transition_Light(
        VI_System_Time := VI_System_Time_MS,
        VI_Start_Time := VI_System_Time_MS,
        VI_Duration := 5000, // 5 секунд на плавное изменение света
        VI_Start_Value := TO_REAL(L_Base_Light),
        VI_End_Value := TO_REAL(L_Target_Base_Light)
    );
    L_Transition_Blinds(
        VI_System_Time := VI_System_Time_MS,
        VI_Start_Time := VI_System_Time_MS,
        VI_Duration := 10000, // 10 секунд на плавное изменение штор
        VI_Start_Value := TO_REAL(L_Base_Blinds),
        VI_End_Value := TO_REAL(L_Target_Base_Blinds)
    );
    L_Prev_Scenario := L_Effective_Scenario;
ELSE
    L_Transition_Light(
        VI_System_Time := VI_System_Time_MS,
        VI_Start_Time := L_Transition_Light.VI_Start_Time,
        VI_Duration := L_Transition_Light.VI_Duration,
        VI_Start_Value := L_Transition_Light.VI_Start_Value,
        VI_End_Value := TO_REAL(L_Target_Base_Light)
    );
    L_Transition_Blinds(
        VI_System_Time := VI_System_Time_MS,
        VI_Start_Time := L_Transition_Blinds.VI_Start_Time,
        VI_Duration := L_Transition_Blinds.VI_Duration,
        VI_Start_Value := L_Transition_Blinds.VI_Start_Value,
        VI_End_Value := TO_REAL(L_Target_Base_Blinds)
    );
END_IF;

L_Base_Light := TO_BYTE(L_Transition_Light.VO_Current_Value);
L_Base_Blinds := TO_BYTE(L_Transition_Blinds.VO_Current_Value);

// 2. Управление освещением
FOR L_i := 1 TO 32 DO
    L_Rule_Light_Active := FALSE;
    L_Rule_Light_Val := 0;
    
    // Проверка правил
    FOR L_j := 1 TO GVL_CONSTANTS.C_MAX_RULES DO
        IF VI_Rule_Actions[L_j].Active AND VI_Rule_Actions[L_j].Target_ID = L_i THEN
            IF VI_Rule_Actions[L_j].Action_Type = E_Rule_Action_Type.ACTION_SET_LIGHTING_BASE THEN
                L_Rule_Light_Active := TRUE;
                L_Rule_Light_Val := REAL_TO_BYTE(VI_Rule_Actions[L_j].Value);
                L_Light_States[L_i] := (L_Rule_Light_Val > 0);
            ELSIF VI_Rule_Actions[L_j].Action_Type = E_Rule_Action_Type.ACTION_TOGGLE_LIGHTING AND VI_Rule_Actions[L_j].Triggered THEN
                L_Light_States[L_i] := NOT L_Light_States[L_i];
            END_IF;
        END_IF;
    END_FOR;

    // Приоритет 1: Физические выключатели (ТЗ 1.0)
    IF VI_Physical_Switches[L_i] AND NOT L_Prev_Switches[L_i] THEN
        L_Light_States[L_i] := NOT L_Light_States[L_i];
        L_Manual_Override[L_i] := TRUE; // Запоминаем ручное переопределение
    END_IF;
    L_Prev_Switches[L_i] := VI_Physical_Switches[L_i];

    // Приоритет 2: Датчики движения (ТЗ 2.0)
    // Защита от дребезга и удержание сигнала движения с помощью TOF
    L_Motion_Timers[L_i](IN := VI_Motion_Sensors[L_i], PT := T#5m, VI_System_Time_MS := VI_System_Time_MS);
    
    // Сброс ручного переопределения, когда комната становится пустой (задний фронт таймера движения)
    IF L_Prev_Motion_Q[L_i] AND NOT L_Motion_Timers[L_i].Q THEN
        L_Manual_Override[L_i] := FALSE;
    END_IF;
    L_Prev_Motion_Q[L_i] := L_Motion_Timers[L_i].Q;

    IF L_Motion_Timers[L_i].Q THEN
        IF NOT L_Manual_Override[L_i] THEN
            L_Light_States[L_i] := TRUE;
        END_IF;
    ELSE
        // Выключаем свет только если нет ручного переопределения
        IF NOT L_Manual_Override[L_i] THEN
            L_Light_States[L_i] := FALSE;
        END_IF;
    END_IF;

    // Приоритет 3: Симуляция (только в режиме Away)
    IF L_Effective_Scenario = E_SCENARIO_TYPE.SCENARIO_AWAY AND L_Effective_Simulation_Active THEN
        L_Light_States[L_i] := VI_Simulation_Lights[L_i];
    END_IF;

    // Приоритет 4: Ручное управление и правила
    IF VI_Manual_Light_Override[L_i] > 0 THEN
        VO_Lighting_Levels[L_i] := VI_Manual_Light_Override[L_i];
    ELSIF L_Rule_Light_Active THEN
        VO_Lighting_Levels[L_i] := L_Rule_Light_Val;
    ELSE
        VO_Lighting_Levels[L_i] := SEL(L_Light_States[L_i], 0, L_Base_Light);
    END_IF;
    
    // 5. Мокрые зоны
    IF VI_Wet_Zone_Map[L_i] AND L_Wet_Zone_Idx <= GVL_CONSTANTS.C_MAX_WET_ZONES THEN
        VO_Wet_Zone_Light_Active[L_Wet_Zone_Idx] := (VO_Lighting_Levels[L_i] > 10);
        L_Wet_Zone_Idx := L_Wet_Zone_Idx + 1;
    END_IF;
END_FOR;

// 3. Управление шторами
FOR L_i := 1 TO GVL_CONSTANTS.C_MAX_BLINDS DO
    L_Rule_Blinds_Active := FALSE;
    L_Rule_Blinds_Val := 0;
    
    // Проверка правил
    FOR L_j := 1 TO GVL_CONSTANTS.C_MAX_RULES DO
        IF VI_Rule_Actions[L_j].Active AND VI_Rule_Actions[L_j].Target_ID = L_i THEN
            IF VI_Rule_Actions[L_j].Action_Type = E_Rule_Action_Type.ACTION_SET_BLINDS THEN
                L_Rule_Blinds_Active := TRUE;
                L_Rule_Blinds_Val := REAL_TO_BYTE(VI_Rule_Actions[L_j].Value);
            END_IF;
        END_IF;
    END_FOR;

    // Приоритет 1: Ручное управление
    IF VI_Manual_Blinds_Override[L_i] > 0 THEN
        VO_Blinds_Positions[L_i] := VI_Manual_Blinds_Override[L_i];
    // Приоритет 2: Правила
    ELSIF L_Rule_Blinds_Active THEN
        VO_Blinds_Positions[L_i] := L_Rule_Blinds_Val;
    // Приоритет 3: Сценарий
    ELSE
        VO_Blinds_Positions[L_i] := L_Base_Blinds;
    END_IF;
END_FOR;

// ========================================
// Lighting V2 shadow execution (phase2)
// ========================================
fbLightingV2Staging(
    VI_Zone_ID := 1,
    VI_Enable := (VO_Lighting_Levels[1] > 0),
    VI_Brightness_Setpoint := BYTE_TO_REAL(VO_Lighting_Levels[1]),
    VI_Scene_ID := TO_INT(L_Effective_Scenario),
    VI_Manual_Override := (VI_Manual_Light_Override[1] > 0),
    VI_Transition_Time_MS := 5000,

    VI_Is_Active := (VO_Lighting_Levels[1] > 0),
    VI_Brightness_Actual := BYTE_TO_REAL(VO_Lighting_Levels[1]),
    VI_Motion_Active := VI_Motion_Sensors[1],
    VI_Ambient_Lux := 0.0,
    VI_Alarm_Active := GVL_STATE.G_Lighting_IO_Fault OR GVL_STATE.G_Lighting_Subsystem_Degraded,

    VO_Command_Shadow => L_Lighting_V2_Command_Shadow,
    VO_State_Shadow => L_Lighting_V2_State_Shadow
);

// ========================================
// Lighting V2 shadow validation
// ========================================
IF ABS(BYTE_TO_REAL(VO_Lighting_Levels[1]) - L_Lighting_V2_Command_Shadow.Brightness_Setpoint) > 0.1 THEN
    L_Lighting_V2_Shadow_Diff_Found := TRUE;
END_IF;
IF ABS(BYTE_TO_REAL(VO_Lighting_Levels[1]) - L_Lighting_V2_State_Shadow.Brightness_Actual) > 0.1 THEN
    L_Lighting_V2_Shadow_Diff_Found := TRUE;
END_IF;
IF VI_Motion_Sensors[1] <> L_Lighting_V2_State_Shadow.Motion_Active THEN
    L_Lighting_V2_Shadow_Diff_Found := TRUE;
END_IF;

// Guarded Lighting V2 enable
IF L_Lighting_V2_Switch_Enabled THEN
    IF NOT L_Lighting_V2_Shadow_Diff_Found THEN
        L_Lighting_V2_Path_Ready := TRUE;
        L_Lighting_Using_Legacy_Fallback := FALSE;
    ELSE
        L_Lighting_V2_Path_Ready := FALSE;
        L_Lighting_Using_Legacy_Fallback := TRUE;
    END_IF;
ELSE
    L_Lighting_V2_Path_Ready := FALSE;
    L_Lighting_Using_Legacy_Fallback := TRUE;
END_IF;



// ========================================
// Blinds V2 shadow execution (phase2)
// ========================================
fbBlindsV2Staging(
    VI_Blind_ID := 1,
    VI_Enable := TRUE,
    VI_Position_Setpoint := VO_Blinds_Positions[1],
    VI_Manual_Override := (VI_Manual_Blinds_Override[1] > 0),
    VI_Scenario_ID := TO_INT(L_Effective_Scenario),
    VI_Safety_Mode := FALSE,

    VI_Position_Actual := VO_Blinds_Positions[1],
    VI_Manual_Override_Active := (VI_Manual_Blinds_Override[1] > 0),
    VI_Is_Moving := FALSE,
    VI_Alarm_Active := GVL_STATE.G_Lighting_IO_Fault,

    VO_Command_Shadow => L_Blinds_V2_Command_Shadow,
    VO_State_Shadow => L_Blinds_V2_State_Shadow
);

// Blinds validation
IF VO_Blinds_Positions[1] <> L_Blinds_V2_Command_Shadow.Position_Setpoint THEN
    L_Blinds_V2_Shadow_Diff_Found := TRUE;
END_IF;
IF VO_Blinds_Positions[1] <> L_Blinds_V2_State_Shadow.Position_Actual THEN
    L_Blinds_V2_Shadow_Diff_Found := TRUE;
END_IF;


// Guarded Blinds V2 enable
IF L_Blinds_V2_Switch_Enabled THEN
    IF NOT L_Blinds_V2_Shadow_Diff_Found THEN
        L_Blinds_V2_Path_Ready := TRUE;
        L_Blinds_Using_Legacy_Fallback := FALSE;
    ELSE
        L_Blinds_V2_Path_Ready := FALSE;
        L_Blinds_Using_Legacy_Fallback := TRUE;
    END_IF;
ELSE
    L_Blinds_V2_Path_Ready := FALSE;
    L_Blinds_Using_Legacy_Fallback := TRUE;
END_IF;

// >>> BULK_SYNC_ANCHOR: FB_Lighting_Blinds_Manager <<<
          
END_FUNCTION_BLOCK

FUNCTION_BLOCK FB_System_Health
  VAR_INPUT
    VI_Smoke_Detected : BOOL;
    VI_Gas_Detected : BOOL;
    VI_CO_Warning_Level : BOOL;
    VI_CO_Alarm_Level : BOOL;
    VI_Leak_Detected : BOOL;
    VI_Sensor_Fault : BOOL := FALSE;
    VI_IO_Offline : BOOL := FALSE;
    VI_Comm_Fault : BOOL := FALSE;
    VI_Watchdog_Fault : BOOL := FALSE;
    VI_Subsystem_Fault : BOOL := FALSE;
  END_VAR
  VAR_OUTPUT
    VO_System_Severity : E_System_Severity;
    VO_Root_Cause : E_System_Root_Cause;
    VO_Sensor_Fault : BOOL;
    VO_IO_Fault : BOOL;
    VO_Comm_Fault : BOOL;
    VO_Subsystem_Degraded : BOOL;
    VO_First_Fault_Active : BOOL;
    VO_First_Fault_Type : INT;
    VO_First_Fault_Source : INT;
  END_VAR

            VO_Sensor_Fault := VI_Sensor_Fault;
VO_IO_Fault := VI_IO_Offline;
VO_Comm_Fault := VI_Comm_Fault;
VO_Subsystem_Degraded := VI_Subsystem_Fault;

VO_System_Severity := E_System_Severity.SEV_NORMAL;
VO_Root_Cause := E_System_Root_Cause.ROOT_NONE;
VO_First_Fault_Active := FALSE;
VO_First_Fault_Type := 0;
VO_First_Fault_Source := 0;

// Priority: FIRE > GAS > CO > WATER > diagnostics
IF VI_Smoke_Detected THEN
    VO_System_Severity := E_System_Severity.SEV_CRITICAL;
    VO_Root_Cause := E_System_Root_Cause.ROOT_FIRE;
    VO_First_Fault_Active := TRUE;
    VO_First_Fault_Type := 5;

ELSIF VI_Gas_Detected THEN
    VO_System_Severity := E_System_Severity.SEV_CRITICAL;
    VO_Root_Cause := E_System_Root_Cause.ROOT_GAS_LEAK;
    VO_First_Fault_Active := TRUE;
    VO_First_Fault_Type := 6;

ELSIF VI_CO_Alarm_Level THEN
    VO_System_Severity := E_System_Severity.SEV_CRITICAL;
    VO_Root_Cause := E_System_Root_Cause.ROOT_CO_CRITICAL;
    VO_First_Fault_Active := TRUE;
    VO_First_Fault_Type := 7;

ELSIF VI_CO_Warning_Level THEN
    VO_System_Severity := E_System_Severity.SEV_WARNING;
    VO_Root_Cause := E_System_Root_Cause.ROOT_CO_WARNING;
    VO_First_Fault_Active := TRUE;
    VO_First_Fault_Type := 7;

ELSIF VI_Leak_Detected THEN
    VO_System_Severity := E_System_Severity.SEV_WARNING;
    VO_Root_Cause := E_System_Root_Cause.ROOT_WATER_LEAK;
    VO_First_Fault_Active := TRUE;
    VO_First_Fault_Type := 8;

ELSIF VI_Watchdog_Fault THEN
    VO_System_Severity := E_System_Severity.SEV_CRITICAL;
    VO_Root_Cause := E_System_Root_Cause.ROOT_WATCHDOG_FAULT;
    VO_First_Fault_Active := TRUE;
    VO_First_Fault_Type := 9;

ELSIF VI_IO_Offline THEN
    VO_System_Severity := E_System_Severity.SEV_DEGRADED;
    VO_Root_Cause := E_System_Root_Cause.ROOT_IO_OFFLINE;
    VO_First_Fault_Active := TRUE;
    VO_First_Fault_Type := 1;

ELSIF VI_Comm_Fault THEN
    VO_System_Severity := E_System_Severity.SEV_DEGRADED;
    VO_Root_Cause := E_System_Root_Cause.ROOT_COMM_FAULT;
    VO_First_Fault_Active := TRUE;
    VO_First_Fault_Type := 3;

ELSIF VI_Sensor_Fault THEN
    VO_System_Severity := E_System_Severity.SEV_DEGRADED;
    VO_Root_Cause := E_System_Root_Cause.ROOT_SENSOR_FAULT;
    VO_First_Fault_Active := TRUE;
    VO_First_Fault_Type := 2;

ELSIF VI_Subsystem_Fault THEN
    VO_System_Severity := E_System_Severity.SEV_DEGRADED;
    VO_Root_Cause := E_System_Root_Cause.ROOT_SUBSYSTEM_FAULT;
    VO_First_Fault_Active := TRUE;
    VO_First_Fault_Type := 4;
END_IF;
// >>> BULK_SYNC_ANCHOR: FB_System_Health <<<
          
END_FUNCTION_BLOCK

FUNCTION_BLOCK FB_DHW_V2_Staging
  VAR_INPUT
    VI_Tank_ID : INT;
    VI_Enable : BOOL;
    VI_Target_Temp : REAL;
    VI_Pump_Enable : BOOL;
    VI_Heating_Priority : BOOL;
    VI_Is_Active : BOOL;
    VI_Tank_Temp : REAL;
    VI_Supply_Temp : REAL;
    VI_Return_Temp : REAL;
    VI_Pump_Actual : BOOL;
    VI_Alarm_Active : BOOL;
  END_VAR
  VAR_OUTPUT
    VO_Command_Shadow : ST_DHW_Command_V2;
    VO_State_Shadow : ST_DHW_State_V2;
  END_VAR

            IF VI_Pump_Enable THEN
    VO_Command_Shadow.Pump_Enable := 1.0;
ELSE
    VO_Command_Shadow.Pump_Enable := 0.0;
END_IF;

VO_State_Shadow.Tank_Temp := VI_Tank_Temp;
VO_State_Shadow.Supply_Temp := VI_Supply_Temp;
          
END_FUNCTION_BLOCK

FUNCTION_BLOCK FB_TwoFactor_Auth
  VAR_INPUT
    VI_System_Time_MS : UDINT;
    VI_Start_Auth : BOOL;
    VI_Method : E_TwoFactor_Method;
    VI_User_Code : STRING(6);
    VI_Reset_Success : BOOL;
  END_VAR
  VAR_OUTPUT
    VO_State : ST_TwoFactor_Auth_State;
    VO_Send_Code_Req : BOOL;
    VO_Code_To_Send : STRING(6);
  END_VAR
  VAR
    L_Generated_Code : STRING(6) := '';
    L_Start_Time : UDINT;
    R_Trig_Start : R_TRIG;
    L_Prev_User_Code : STRING(6);
    L_Lockout_Start_Time : UDINT;
    fbHMAC : FB_HMAC_SHA1;
    L_Elapsed_Time : UDINT;
    L_Time_Step : UDINT;
    L_Message : ARRAY[0..7] OF BYTE;
    L_Key : ARRAY[0..63] OF BYTE;
    L_Offset : INT;
    L_Truncated_Hash : UDINT;
    L_i : INT;
    L_Current_TOTP : STRING(6);
    L_Prev_TOTP : STRING(6);
    L_Code_Valid : BOOL;
  END_VAR

            R_Trig_Start(CLK := VI_Start_Auth);

IF VI_Reset_Success THEN
    VO_State.Is_Success := FALSE;
END_IF;

IF R_Trig_Start.Q AND NOT VO_State.is_pending AND NOT VO_State.Is_Locked THEN
    VO_State.is_pending := TRUE;
    VO_State.Auth_Method := VI_Method;
    L_Start_Time := VI_System_Time_MS;
    VO_State.Attempts_Left := 3;
    VO_State.Is_Success := FALSE;
    VO_State.Is_Locked := FALSE;
    L_Prev_User_Code := '';
    
    IF VI_Method <> E_TwoFactor_Method.TF_METHOD_TOTP THEN
        // Генерируем одноразовый код через HMAC (без упрощенного алгоритма "по времени")
        L_Time_Step := VI_System_Time_MS / 30000;
        L_Key[0] := 16#31; L_Key[1] := 16#32; L_Key[2] := 16#33; L_Key[3] := 16#34; // Секрет-шаблон, заменяется из конфигурации
        FOR L_i := 0 TO 7 DO L_Message[7 - L_i] := TO_BYTE(SHR(L_Time_Step + L_Start_Time, L_i * 8) AND 16#FF); END_FOR;
        fbHMAC(Key := L_Key, KeyLength := 4, Message := L_Message, MessageLength := 8);
        L_Offset := TO_INT(fbHMAC.Hash[19] AND 16#0F);
        L_Truncated_Hash := (SHL(TO_UDINT(fbHMAC.Hash[L_Offset] AND 16#7F), 24) OR SHL(TO_UDINT(fbHMAC.Hash[L_Offset+1] AND 16#FF), 16) OR SHL(TO_UDINT(fbHMAC.Hash[L_Offset+2] AND 16#FF), 8) OR TO_UDINT(fbHMAC.Hash[L_Offset+3] AND 16#FF));
        L_Generated_Code := UDINT_TO_STRING(L_Truncated_Hash MOD 1000000);
        WHILE LEN(L_Generated_Code) < 6 DO
            L_Generated_Code := CONCAT('0', L_Generated_Code);
        END_WHILE;
        
        VO_Code_To_Send := L_Generated_Code;
        VO_Send_Code_Req := TRUE;
    ELSE
        // Для TOTP код не отправляем
        VO_Code_To_Send := '';
        VO_Send_Code_Req := FALSE;
    END_IF;
ELSE
    VO_Send_Code_Req := FALSE;
END_IF;

IF VO_State.is_pending THEN
    L_Elapsed_Time := (SEL(VI_System_Time_MS >= L_Start_Time, VI_System_Time_MS - L_Start_Time, (4294967295 - L_Start_Time) + VI_System_Time_MS + 1));

    IF L_Elapsed_Time < (GVL_CONSTANTS.C_MS_IN_MINUTE * 5) THEN
        VO_State.Time_Left_S := TO_UINT(((GVL_CONSTANTS.C_MS_IN_MINUTE * 5) - L_Elapsed_Time) / 1000);
    ELSE
        VO_State.Time_Left_S := 0;
    END_IF;
    
    IF VI_User_Code <> '' AND VI_User_Code <> L_Prev_User_Code THEN
        L_Code_Valid := FALSE;
        
        IF VI_Method = E_TwoFactor_Method.TF_METHOD_TOTP THEN
            // Вычисляем TOTP для текущего шага времени (30 секунд)
            L_Time_Step := VI_System_Time_MS / 30000; 
            
            // Подготовка ключа (в реальном проекте берется из GVL_CONFIG)
            L_Key[0] := 16#31; L_Key[1] := 16#32; L_Key[2] := 16#33; L_Key[3] := 16#34; // '1234'
            
            // Проверка текущего шага
            FOR L_i := 0 TO 7 DO L_Message[7 - L_i] := TO_BYTE(SHR(L_Time_Step, L_i * 8) AND 16#FF); END_FOR;
            fbHMAC(Key := L_Key, KeyLength := 4, Message := L_Message, MessageLength := 8);
            L_Offset := TO_INT(fbHMAC.Hash[19] AND 16#0F);
            L_Truncated_Hash := (SHL(TO_UDINT(fbHMAC.Hash[L_Offset] AND 16#7F), 24) OR SHL(TO_UDINT(fbHMAC.Hash[L_Offset+1] AND 16#FF), 16) OR SHL(TO_UDINT(fbHMAC.Hash[L_Offset+2] AND 16#FF), 8) OR TO_UDINT(fbHMAC.Hash[L_Offset+3] AND 16#FF));
            L_Current_TOTP := UDINT_TO_STRING(L_Truncated_Hash MOD 1000000);
            WHILE LEN(L_Current_TOTP) < 6 DO L_Current_TOTP := CONCAT('0', L_Current_TOTP); END_WHILE;
            
            // Проверка предыдущего шага (для компенсации рассинхронизации)
            FOR L_i := 0 TO 7 DO L_Message[7 - L_i] := TO_BYTE(SHR(L_Time_Step - 1, L_i * 8) AND 16#FF); END_FOR;
            fbHMAC(Key := L_Key, KeyLength := 4, Message := L_Message, MessageLength := 8);
            L_Offset := TO_INT(fbHMAC.Hash[19] AND 16#0F);
            L_Truncated_Hash := (SHL(TO_UDINT(fbHMAC.Hash[L_Offset] AND 16#7F), 24) OR SHL(TO_UDINT(fbHMAC.Hash[L_Offset+1] AND 16#FF), 16) OR SHL(TO_UDINT(fbHMAC.Hash[L_Offset+2] AND 16#FF), 8) OR TO_UDINT(fbHMAC.Hash[L_Offset+3] AND 16#FF));
            L_Prev_TOTP := UDINT_TO_STRING(L_Truncated_Hash MOD 1000000);
            WHILE LEN(L_Prev_TOTP) < 6 DO L_Prev_TOTP := CONCAT('0', L_Prev_TOTP); END_WHILE;
            
            IF VI_User_Code = L_Current_TOTP OR VI_User_Code = L_Prev_TOTP THEN
                L_Code_Valid := TRUE;
            END_IF;
        ELSE
            IF VI_User_Code = L_Generated_Code THEN
                L_Code_Valid := TRUE;
            END_IF;
        END_IF;
        
        IF L_Code_Valid THEN
            VO_State.Is_Success := TRUE;
            VO_State.is_pending := FALSE;
        ELSE
            IF VO_State.Attempts_Left > 0 THEN
                VO_State.Attempts_Left := VO_State.Attempts_Left - 1;
            END_IF;
            
            IF VO_State.Attempts_Left = 0 THEN
                VO_State.Is_Locked := TRUE;
                VO_State.is_pending := FALSE;
                L_Lockout_Start_Time := VI_System_Time_MS; // Блокировка на 5 минут
            END_IF;
        END_IF;
    END_IF;
    L_Prev_User_Code := VI_User_Code;
    
    IF L_Elapsed_Time > (GVL_CONSTANTS.C_MS_IN_MINUTE * 5) THEN
        VO_State.is_pending := FALSE; // Таймаут
    END_IF;
END_IF;

IF VO_State.Is_Locked THEN
    IF (SEL(VI_System_Time_MS >= L_Lockout_Start_Time, VI_System_Time_MS - L_Lockout_Start_Time, (4294967295 - L_Lockout_Start_Time) + VI_System_Time_MS + 1)) >= (GVL_CONSTANTS.C_MS_IN_MINUTE * 5) THEN
        VO_State.Is_Locked := FALSE;
    END_IF;
END_IF;
          
END_FUNCTION_BLOCK

FUNCTION_BLOCK FB_CO_Detector
  VAR_INPUT
    VI_CO_PPM : REAL;
    VI_Threshold_Warning : REAL := 30.0;
    VI_Threshold_Alarm : REAL := 70.0;
  END_VAR
  VAR_OUTPUT
    VO_CO_Warning_Level : BOOL;
    VO_CO_Alarm_Level : BOOL;
  END_VAR

            VO_CO_Warning_Level := (VI_CO_PPM >= VI_Threshold_Warning);
VO_CO_Alarm_Level   := (VI_CO_PPM >= VI_Threshold_Alarm);
          
END_FUNCTION_BLOCK

FUNCTION_BLOCK FB_System_Timer
  VAR_INPUT
    IN : BOOL;
    PT : TIME;
    VI_System_Time_MS : UDINT;
  END_VAR
  VAR_OUTPUT
    Q : BOOL;
    ET : TIME;
  END_VAR
  VAR
    L_Start_Time : UDINT;
    L_Running : BOOL;
  END_VAR

            // ==============================================================================
// Блок таймера, привязанный к системному времени (System Timer)
// Назначение:
// - Замена стандартного TON для обеспечения точной выдержки времени,
//   независимой от времени цикла ПЛК, с использованием единого системного времени.
// ==============================================================================



IF IN THEN
    IF NOT L_Running THEN
        L_Start_Time := VI_System_Time_MS;
        L_Running := TRUE;
        ET := T#0s;
        Q := FALSE;
    ELSE
        // Обработка переполнения UDINT (примерно 49 дней)
        ET := TO_TIME((SEL(VI_System_Time_MS >= L_Start_Time, VI_System_Time_MS - L_Start_Time, (4294967295 - L_Start_Time) + VI_System_Time_MS + 1)));
        
        IF ET >= PT THEN
            Q := TRUE;
            ET := PT;
        ELSE
            Q := FALSE;
        END_IF;
    END_IF;
ELSE
    L_Running := FALSE;
    ET := T#0s;
    Q := FALSE;
END_IF;
// >>> BULK_SYNC_ANCHOR: FB_System_Timer <<<
          
END_FUNCTION_BLOCK

FUNCTION_BLOCK FB_PLC_Heartbeat
  VAR_INPUT
    VI_Local_ID : BYTE;
    VI_System_Time : UDINT;
    VI_Remote_Pulse : BOOL;
    VI_Remote_Is_Active : BOOL;
    VI_Gateway_Ping_OK : BOOL;
  END_VAR
  VAR_OUTPUT
    VO_Is_Active : BOOL;
    VO_RTT_MS : UDINT;
    VO_Loss_Count : UDINT;
    VO_Max_RTT : UDINT;
  END_VAR
  VAR
    L_Last_Pulse : BOOL;
    L_Last_Pulse_Time : UDINT;
    L_Timeout : UDINT := 500;
    L_Pulse_Send_Time : UDINT;
    L_Last_Loss_Time : UDINT;
    L_Elapsed_Time : UDINT;
  END_VAR

            // Вспомогательная функция для безопасного вычисления разницы времени
L_Elapsed_Time := (VI_System_Time - L_Last_Pulse_Time);

// 1. Мониторинг "сердцебиения" и расчет сетевых задержек (ТЗ 8.4)
IF VI_Remote_Pulse <> L_Last_Pulse THEN
    // Вычисляем время между изменениями сигнала
    VO_RTT_MS := L_Elapsed_Time;
    // Фиксируем пиковые задержки для диагностики сети
    IF VO_RTT_MS > VO_Max_RTT THEN VO_Max_RTT := VO_RTT_MS; END_IF;
    L_Last_Pulse := VI_Remote_Pulse;
    L_Last_Pulse_Time := VI_System_Time;
    L_Elapsed_Time := 0; // Сбрасываем после обновления
END_IF;

// Подсчет статистики потерь связи (ТЗ 8.4)
IF L_Elapsed_Time > L_Timeout THEN
    IF (VI_System_Time - L_Last_Loss_Time) >= 1000 THEN
        VO_Loss_Count := VO_Loss_Count + 1;
        L_Last_Loss_Time := VI_System_Time;
    END_IF;
ELSE
    L_Last_Loss_Time := VI_System_Time;
END_IF;

// 2. Логика определения роли (Active/Standby) и предотвращение Split-Brain (ТЗ 8.3)
// Уровень 1: Проверка наличия связи с партнером
IF L_Elapsed_Time < L_Timeout THEN
    // Связь есть: Договариваемся о ролях на основе приоритета ID
    IF VI_Local_ID = 1 THEN
        VO_Is_Active := TRUE; // ПЛК А всегда активен при наличии связи
    ELSE
        VO_Is_Active := NOT VI_Remote_Is_Active; // ПЛК B активен только если А не активен
    END_IF;
ELSE
    // Связи нет: Пытаемся определить, кто из нас "живее"
    // Уровень 3: Если связи с партнером нет, проверяем доступность внешнего шлюза
    IF VI_Local_ID = 1 THEN
        // ПЛК А становится активным всегда при потере связи с партнером (fallback)
        VO_Is_Active := TRUE;
    ELSE
        // ПЛК B ждет таймаут удержания роли (2 секунды), прежде чем стать активным
        IF L_Elapsed_Time >= 2000 THEN
            // ПЛК B берет управление если он видит шлюз, а связи с А нет.
            // Если шлюз недоступен, B ждет дольше (fallback).
            IF VI_Gateway_Ping_OK THEN
                VO_Is_Active := TRUE;
            ELSIF L_Elapsed_Time >= 5000 THEN
                VO_Is_Active := TRUE; // Fallback: ПЛК А мертв и шлюз мертв
            ELSE
                VO_Is_Active := FALSE;
            END_IF;
        ELSE
            VO_Is_Active := FALSE;
        END_IF;
    END_IF;
END_IF;
          
END_FUNCTION_BLOCK

FUNCTION_BLOCK FB_Device_Predictive_Diag
  VAR_INPUT
    VI_Current_Value : REAL;
    VI_Nominal_Value : REAL;
    VI_Is_Running : BOOL;
    VI_Reset_Stats : BOOL;
    VI_System_Time_MS : UDINT;
  END_VAR
  VAR_IN_OUT
    VIO_Health_Data : ST_Device_Health;
  END_VAR
  VAR
    L_Prev_Running : BOOL;
    L_Start_Time : UDINT;
    L_Last_Calc_Time : UDINT;
    L_Elapsed_MS : UDINT;
    L_Accumulated_MS : UDINT;
    L_Timer_Running : FB_System_Timer;
  END_VAR

            // 0. Сброс статистики
IF VI_Reset_Stats THEN
    VIO_Health_Data.Starts_Count := 0;
    VIO_Health_Data.Sample_Count := 0;
    VIO_Health_Data.Current_Sum := 0.0;
    VIO_Health_Data.Avg_Start_Current := 0.0;
    VIO_Health_Data.Health_Score := 100;
    VIO_Health_Data.Maintenance_Required := FALSE;
    VIO_Health_Data.Warning_Message := '';
    VIO_Health_Data.Last_Start_Current := 0.0;
    VIO_Health_Data.Total_Runtime_Hours := 0;
    L_Accumulated_MS := 0;
END_IF;

// 1. Счётчик пусков и замер пускового тока
IF VI_Is_Running AND NOT L_Prev_Running THEN
    VIO_Health_Data.Starts_Count := VIO_Health_Data.Starts_Count + 1;
    VIO_Health_Data.Last_Start_Current := VI_Current_Value;
    L_Start_Time := VI_System_Time_MS;
    L_Last_Calc_Time := VI_System_Time_MS;
    
    // Обновление среднего пускового тока
    VIO_Health_Data.Sample_Count := VIO_Health_Data.Sample_Count + 1;
    VIO_Health_Data.Current_Sum := VIO_Health_Data.Current_Sum + VI_Current_Value;
    VIO_Health_Data.Avg_Start_Current := VIO_Health_Data.Current_Sum / UDINT_TO_REAL(VIO_Health_Data.Sample_Count);
    
    // 2. Анализ отклонения пускового тока (п. 12.1 ТЗ)
    IF VI_Current_Value > (VI_Nominal_Value * 1.5) THEN
        VIO_Health_Data.Health_Score := TO_BYTE(LIMIT(0, TO_INT(VIO_Health_Data.Health_Score) - 5, 100));
    ELSIF VI_Current_Value > (VI_Nominal_Value * 1.2) THEN
        VIO_Health_Data.Health_Score := TO_BYTE(LIMIT(0, TO_INT(VIO_Health_Data.Health_Score) - 1, 100));
    ELSIF VI_Current_Value < (VI_Nominal_Value * 0.5) THEN
        VIO_Health_Data.Health_Score := TO_BYTE(LIMIT(0, TO_INT(VIO_Health_Data.Health_Score) - 2, 100));
    END_IF;
END_IF;

// 3. Анализ рабочего тока и наработки
IF VI_Is_Running THEN
    L_Elapsed_MS := (VI_System_Time_MS - L_Last_Calc_Time);
    L_Accumulated_MS := L_Accumulated_MS + L_Elapsed_MS;
    L_Last_Calc_Time := VI_System_Time_MS;
    
    // Обновляем наработку каждый час (3600000 мс)
    IF L_Accumulated_MS >= 3600000 THEN
        VIO_Health_Data.Total_Runtime_Hours := VIO_Health_Data.Total_Runtime_Hours + 1;
        L_Accumulated_MS := L_Accumulated_MS - 3600000;
        
        // Естественный износ: -1% здоровья каждые 1000 часов
        IF (VIO_Health_Data.Total_Runtime_Hours MOD 1000) = 0 THEN
            VIO_Health_Data.Health_Score := TO_BYTE(LIMIT(0, TO_INT(VIO_Health_Data.Health_Score) - 1, 100));
        END_IF;
        
        // Анализ рабочего тока (после пускового режима)
        IF (VI_System_Time_MS - L_Start_Time) > 10000 THEN // 10 секунд после пуска
            IF VI_Current_Value > (VI_Nominal_Value * 1.1) THEN
                // Повышенный рабочий ток - ускоренный износ (-1% в час)
                VIO_Health_Data.Health_Score := TO_BYTE(LIMIT(0, TO_INT(VIO_Health_Data.Health_Score) - 1, 100));
            END_IF;
        END_IF;
    END_IF;
END_IF;

// 4. Генерация предупреждения
IF VIO_Health_Data.Health_Score < 20 THEN
    VIO_Health_Data.Maintenance_Required := TRUE;
    VIO_Health_Data.Warning_Message := 'Критический износ: проверьте механику';
ELSIF VIO_Health_Data.Health_Score < 60 THEN
    VIO_Health_Data.Maintenance_Required := FALSE;
    VIO_Health_Data.Warning_Message := 'Предупреждение: повышенное трение';
ELSE
    VIO_Health_Data.Maintenance_Required := FALSE;
    VIO_Health_Data.Warning_Message := 'В норме';
END_IF;

L_Prev_Running := VI_Is_Running;
          
END_FUNCTION_BLOCK

FUNCTION_BLOCK FB_Ventilation_V2_Staging
  VAR_INPUT
    VI_Zone_ID : INT;
    VI_Enable : BOOL;
    VI_Fan_Speed_Setpoint : REAL;
    VI_Damper_Position_Setpoint : REAL;
    VI_Heat_Recovery_Enabled : BOOL;
    VI_Is_Active : BOOL;
    VI_Fan_Speed_Actual : REAL;
    VI_Supply_Temp : REAL;
    VI_Extract_Temp : REAL;
    VI_Filter_Dirty : BOOL;
    VI_Alarm_Active : BOOL;
  END_VAR
  VAR_OUTPUT
    VO_Command_Shadow : ST_Ventilation_Command_V2;
    VO_State_Shadow : ST_Ventilation_State_V2;
  END_VAR

            VO_Command_Shadow.Fan_Speed_Setpoint := VI_Fan_Speed_Setpoint;
VO_State_Shadow.Supply_Temp := VI_Supply_Temp;
          
END_FUNCTION_BLOCK

FUNCTION_BLOCK FB_DHW_Manager
  VAR_INPUT
    VI_System_Time_MS : UDINT;
    VI_Current_TOD : TOD;
    VI_IsActivePLC : BOOL;
    VI_Temp : REAL;
    VI_Pressure : REAL;
    VI_Config : ST_DHW_Config;
    VI_Current_Day_Of_Week : UINT;
    VI_Reset_Errors : BOOL;
    VI_Emergency_Stop : BOOL;
    VI_System_Mode : E_System_Operating_Mode;
    VI_IO_Modules_Online : ARRAY[1..GVL_CONSTANTS.C_MAX_MODULES] OF BOOL;
  END_VAR
  VAR_OUTPUT
    VO_Status : ST_DHW_Status;
    VO_Heating_Pump : BOOL;
    VO_Circ_Pump : BOOL;
  END_VAR
  VAR
    fbDHWV2Staging : FB_DHW_V2_Staging;
    L_DHW_V2_Command_V2 : ST_DHW_Command_V2;
    L_DHW_V2_State_V2 : ST_DHW_State_V2;
    L_DHW_V2_Shadow_Diff_Found : BOOL;
    L_DHW_V2_Switch_Enabled : BOOL;
    L_DHW_V2_Path_Ready : BOOL;
    L_DHW_Using_Legacy_Fallback : BOOL;
    L_i : INT;
    L_Current_TOD : TOD;
    L_Legionella_Active : BOOL;
    L_Legionella_Timer : FB_System_Timer;
    L_Last_Good_Temp : REAL := 55.0;
    L_Legionella_Done_Today : BOOL;
    L_Last_Legionella_Day : UINT;
    fbTempValidator : FB_Analog_Validator;
    fbPressValidator : FB_Analog_Validator;
    L_Error_Latched : BOOL;
    L_Error_ID_Latched : WORD;
    L_Policy_Degraded : BOOL;
    L_Policy_Freeze_Protection : BOOL;
    L_Policy_Safe_Stop : BOOL;
    L_Target_Temp_Adjusted : REAL;
  END_VAR

            // >>> SYNC_TEST_MARKER_001 <<<


IF NOT VI_IsActivePLC THEN RETURN; END_IF;

L_DHW_V2_Shadow_Diff_Found := FALSE;
L_DHW_V2_Switch_Enabled := TRUE;
L_DHW_V2_Path_Ready := FALSE;
L_DHW_Using_Legacy_Fallback := TRUE;

GVL_STATE.G_DHW_IO_Fault := FALSE;
GVL_STATE.G_DHW_Sensor_Fault := FALSE;
GVL_STATE.G_DHW_Subsystem_Degraded := FALSE;

IF VI_Emergency_Stop THEN
    VO_Heating_Pump := FALSE;
    VO_Circ_Pump := FALSE;
    VO_Status.Warning := FALSE;
    VO_Status.Error := TRUE;
    VO_Status.Error_ID := TO_WORD(GVL_CONFIG.ERR_DHW_IO_OFFLINE); // временно используем общий аварийный код до детализации safety-кодов
    VO_Status.Heating_Pump_On := FALSE;
    VO_Status.Circ_Pump_On := FALSE;
    RETURN;
END_IF;

// Фиксация текущего времени
L_Current_TOD := VI_Current_TOD;

// ========================================
// DHW POLICY LAYER
// ========================================
L_Policy_Safe_Stop := (VI_System_Mode = E_System_Operating_Mode.MODE_SAFE_STOP);
L_Policy_Freeze_Protection := (VI_System_Mode = E_System_Operating_Mode.MODE_FREEZE_PROTECTION);
L_Policy_Degraded := (VI_System_Mode = E_System_Operating_Mode.MODE_DEGRADED);
L_Target_Temp_Adjusted := VI_Config.Target_Temp;
IF L_Policy_Degraded THEN
    L_Target_Temp_Adjusted := VI_Config.Target_Temp - VI_Config.Degraded_Target_Delta;
END_IF;

// ========================================
// DHW POLICY OVERRIDE
// ========================================
IF L_Policy_Safe_Stop THEN
    VO_Heating_Pump := FALSE;
    VO_Circ_Pump := FALSE;
    RETURN;
END_IF;

IF L_Policy_Freeze_Protection THEN
    VO_Heating_Pump := FALSE;
    VO_Circ_Pump := FALSE;
    RETURN;
END_IF;

// Сброс признака выполнения термодезинфекции при смене дня.
IF L_Last_Legionella_Day <> VI_Current_Day_Of_Week THEN
    L_Legionella_Done_Today := FALSE;
    L_Last_Legionella_Day := VI_Current_Day_Of_Week;
END_IF;

// Базовый сброс незащёлкнутых статусных флагов на текущий цикл.
// Критические ошибки ниже могут зафиксироваться и завершить выполнение через RETURN.
VO_Status.Warning := FALSE;
VO_Status.Error := FALSE;
VO_Status.Error_ID := 0;

// Сброс ошибок
IF VI_Reset_Errors THEN
    L_Error_Latched := FALSE;
    L_Error_ID_Latched := 0;
END_IF;

// Проверка связи с модулями ввода-вывода
FOR L_i := 1 TO GVL_CONSTANTS.C_MAX_MODULES DO
    IF NOT VI_IO_Modules_Online[L_i] THEN
        L_Error_Latched := TRUE;
        GVL_STATE.G_DHW_IO_Fault := TRUE;
        L_Error_ID_Latched := TO_WORD(GVL_CONFIG.ERR_DHW_IO_OFFLINE); // Потеря связи с модулями ввода-вывода
    END_IF;
END_FOR;

// 1. Обработка неисправностей датчиков и сервисных режимов (ТЗ 7.0)
fbTempValidator(
    VI_Value := VI_Temp,
    VI_Min_Valid := 0.0,
    VI_Max_Valid := 100.0,
    VI_Fallback_Mode := 0,
    VI_Default_Value := 55.0
);

fbPressValidator(
    VI_Value := VI_Pressure,
    VI_Min_Valid := 0.0,
    VI_Max_Valid := 10.0,
    VI_Fallback_Mode := 0
);

VO_Status.Temp := fbTempValidator.VO_Value;
VO_Status.Pressure := fbPressValidator.VO_Value;

// Сохраняем последнее достоверное значение температуры ГВС.
// Используется только для диагностики/сервиса, не для fallback-управления.
IF NOT fbTempValidator.VO_Error THEN
    L_Last_Good_Temp := VO_Status.Temp;
END_IF;

IF fbTempValidator.VO_Error THEN
    GVL_STATE.G_DHW_Sensor_Fault := TRUE;
    L_Error_Latched := TRUE;
    L_Error_ID_Latched := TO_WORD(GVL_CONFIG.ERR_DHW_TEMP_SENSOR_FAULT); // Критическая ошибка датчика температуры
ELSIF (VO_Status.Pressure < 1.0 OR VO_Status.Pressure > 4.0) AND NOT fbPressValidator.VO_Error THEN
    L_Error_Latched := TRUE;
    L_Error_ID_Latched := TO_WORD(GVL_CONFIG.ERR_DHW_PRESSURE_OUT_OF_RANGE); // Давление вне нормы
END_IF;

IF L_Error_Latched THEN
    // Критическая ошибка: переход в безопасное состояние с полной остановкой насосов.
    VO_Heating_Pump := FALSE;
    VO_Circ_Pump := FALSE;
    VO_Status.Warning := FALSE;
    VO_Status.Error := TRUE;
    VO_Status.Error_ID := L_Error_ID_Latched;
    VO_Status.Heating_Pump_On := FALSE;
    VO_Status.Circ_Pump_On := FALSE;
    RETURN;
END_IF;

// Ошибка датчика давления не останавливает ГВС,
// но переводит подсистему в режим предупреждения (degraded mode).
IF fbPressValidator.VO_Error THEN
    GVL_STATE.G_DHW_Sensor_Fault := TRUE;
    GVL_STATE.G_DHW_Subsystem_Degraded := TRUE;
    VO_Status.Warning := TRUE;
    VO_Status.Error := FALSE;
    VO_Status.Error_ID := TO_WORD(GVL_CONFIG.ERR_DHW_PRESSURE_SENSOR_FAULT);
END_IF;

// 2. Логика поддержания температуры воды в бойлере (Нагрев)
// На этом этапе FB уже выполняется только на активном ПЛК.
    
// Термическая дезинфекция (Легионелла)
IF VI_Config.Anti_Legionella_Enabled
   AND (VI_Current_Day_Of_Week = VI_Config.Anti_Legionella_Day)
   AND (L_Current_TOD >= TOD#02:00)
   AND (L_Current_TOD <= TOD#04:00)
   AND NOT L_Legionella_Done_Today THEN
    L_Legionella_Active := TRUE;
ELSE
    L_Legionella_Active := FALSE;
END_IF;

L_Legionella_Timer(IN := L_Legionella_Active AND VO_Status.Temp >= 70.0, PT := T#30m, VI_System_Time_MS := VI_System_Time_MS);
IF L_Legionella_Timer.Q THEN
    L_Legionella_Active := FALSE; // Дезинфекция завершена
    L_Legionella_Done_Today := TRUE; // Повторно в те же сутки не запускать
END_IF;

// Двухпозиционное регулирование с гистерезисом
IF L_Legionella_Active THEN
    IF VO_Status.Temp < 70.0 THEN
        VO_Heating_Pump := TRUE;
    ELSIF VO_Status.Temp > 72.0 THEN
        VO_Heating_Pump := FALSE;
    END_IF;
ELSE
    IF VO_Status.Temp < (L_Target_Temp_Adjusted - VI_Config.Hysteresis) THEN
        VO_Heating_Pump := TRUE;
    ELSIF VO_Status.Temp > (L_Target_Temp_Adjusted + VI_Config.Hysteresis) THEN
        VO_Heating_Pump := FALSE;
    END_IF;
END_IF;

// 3. Управление циркуляционным насосом ГВС по расписанию
// Рециркуляция обеспечивает мгновенное наличие горячей воды у потребителя
VO_Circ_Pump := SEL(VI_Config.Circulation_Schedule_Enabled AND NOT (VI_Config.Night_Mode_Enabled AND (L_Current_TOD < VI_Config.Circulation_Start OR L_Current_TOD > VI_Config.Circulation_End)), FALSE, TRUE);

// Формирование статусных данных для визуализации.
// К этому моменту статус уже консистентен:
// - Error = критическая ошибка с остановкой ГВС
// - Warning = деградация без остановки
VO_Status.Heating_Pump_On := VO_Heating_Pump;
VO_Status.Circ_Pump_On := VO_Circ_Pump;

// ========================================
// DHW V2 staging execution
// ========================================
fbDHWV2Staging(
    VI_Tank_ID := 1,
    VI_Enable := TRUE,
    VI_Target_Temp := VI_Config.Target_Temp,
    VI_Pump_Enable := VO_Heating_Pump,
    VI_Heating_Priority := FALSE,

    VI_Is_Active := TRUE,
    VI_Tank_Temp := VO_Status.Temp,
    VI_Supply_Temp := VO_Status.Temp,
    VI_Return_Temp := VO_Status.Temp,
    VI_Pump_Actual := VO_Heating_Pump,
    VI_Alarm_Active := VO_Status.Error,

    VO_Command_Shadow => L_DHW_V2_Command_V2,
    VO_State_Shadow => L_DHW_V2_State_V2
);

// ========================================
// DHW V2 staging validation
// ========================================
IF VO_Heating_Pump <> (L_DHW_V2_Command_V2.Pump_Enable > 0.5) THEN
    L_DHW_V2_Shadow_Diff_Found := TRUE;
END_IF;
IF ABS(VO_Status.Temp - L_DHW_V2_State_V2.Tank_Temp) > 0.1 THEN
    L_DHW_V2_Shadow_Diff_Found := TRUE;
END_IF;
IF ABS(VO_Status.Pressure - L_DHW_V2_State_V2.Supply_Temp) > 0.1 THEN
    L_DHW_V2_Shadow_Diff_Found := TRUE;
END_IF;

// Guarded DHW V2 enable
IF L_DHW_V2_Switch_Enabled THEN
    IF NOT L_DHW_V2_Shadow_Diff_Found THEN
        L_DHW_V2_Path_Ready := TRUE;
        L_DHW_Using_Legacy_Fallback := FALSE;
    ELSE
        L_DHW_V2_Path_Ready := FALSE;
        L_DHW_Using_Legacy_Fallback := TRUE;
    END_IF;
ELSE
    L_DHW_V2_Path_Ready := FALSE;
    L_DHW_Using_Legacy_Fallback := TRUE;
END_IF;

// >>> BULK_SYNC_ANCHOR: FB_DHW_Manager <<<
          
END_FUNCTION_BLOCK

FUNCTION_BLOCK FB_Alarm_Manager
  VAR_INPUT
    VI_System_Time_MS : UDINT;
    VI_IsActivePLC : BOOL;
    VI_Gas_Alarm : BOOL;
    VI_Fire_Alarm : BOOL;
    VI_Flood_Alarm : BOOL;
    VI_Security_Alarm : BOOL;
    VI_First_Fault_Active : BOOL;
    VI_First_Fault_Type : INT;
    VI_First_Fault_Source : INT;
    VI_Security_Msg : STRING(200);
    VI_Acknowledge_All : BOOL;
    VI_Mute_Siren : BOOL;
  END_VAR
  VAR_OUTPUT
    VO_Global_Critical : BOOL;
    VO_Global_Warning : BOOL;
    VO_Siren_Active : BOOL;
    VO_Active_Count : INT;
    VO_Unacked_Count : INT;
    VO_Event_Pulse : BOOL;
    VO_Event_Code : UDINT;
    VO_Event_Value : REAL;
    VO_Alarm_List : ARRAY[1..GVL_CONSTANTS.C_MAX_ALARMS] OF ST_Alarm_Record;
  END_VAR
  VAR_IN_OUT
    VI_Boiler_Errors : ARRAY[1..GVL_CONSTANTS.C_MAX_BOILERS] OF BOOL;
  END_VAR
  VAR_IN_OUT
    VIO_Next_Alarm_ID : UDINT;
  END_VAR
  VAR
    fbCompatAlarm : ARRAY[1..GVL_CONSTANTS.C_MAX_ALARMS] OF FB_Alarm_Compatibility_Package;
    L_i, L_j, L_k : INT;
    L_Target_Slot : INT;
    L_Min_Pri : INT;
    L_Pending_Alarms : ARRAY[1..10] OF ST_Alarm_Record;
    L_Pending_Count : INT := 0;
    T_Debounce_Gas : FB_System_Timer;
    T_Debounce_Fire : FB_System_Timer;
    T_Debounce_Flood : FB_System_Timer;
    T_Debounce_Security : FB_System_Timer;
    R_Trig_Gas : R_TRIG;
    R_Trig_Fire : R_TRIG;
    R_Trig_Flood : R_TRIG;
    R_Trig_Security : R_TRIG;
    R_Trig_First_Fault : R_TRIG;
    R_Trig_Boiler : ARRAY[1..GVL_CONSTANTS.C_MAX_BOILERS] OF R_TRIG;
    L_First_Fault_Source_Text : STRING(32);
    L_First_Fault_Type_Text : STRING(32);
    L_Event_Pulse_Latched : BOOL;
    L_Alarm_Compat_All_OK : BOOL;
    L_Alarm_First_Warning : STRING(255);
    L_Alarm_First_Warning_Latched : BOOL;
    L_Alarm_Shadow_Mismatch : BOOL;
    L_Alarm_Shadow_First_Mismatch : INT;
    L_Alarm_V2_Switch_Enabled : BOOL;
    L_Alarm_V2_Path_Ready : BOOL;
    L_Alarm_Using_Legacy_Fallback : BOOL;
    fbAlarmV2Core : FB_Alarm_V2_Core;
    fbHistoryV2Core : FB_History_V2_Core;
    fbBlackBoxV2Core : FB_BlackBox_V2_Core;
    L_BlackBox_V2_Snapshot_Shadow : ST_BlackBox_Snapshot_V2;
    L_History_V2_Shadow_Diff_Found : BOOL;
    L_History_V2_Shadow_First_Diff_Slot : INT;
    L_BlackBox_V2_Shadow_Diff_Found : BOOL;
    L_History_V2_Buffer_Shadow : ARRAY[1..GVL_CONSTANTS.C_MAX_HISTORY_RECORDS] OF ST_History_Event_V2;
    L_Alarm_V2_Shadow_Compare_Enabled : BOOL;
    L_Alarm_V2_Shadow_Diff_Found : BOOL;
    L_Alarm_V2_Shadow_First_Diff_Slot : INT;
    L_Alarm_V2_Event_Pulse : BOOL;
    L_Alarm_V2_Event_Code : UDINT;
    L_Alarm_V2_Event_Value : REAL;
    L_Alarm_V2_List_Shadow : ARRAY[1..GVL_CONSTANTS.C_MAX_ALARMS] OF ST_Alarm_Record;
    L_Alarm_V2_Next_ID_Shadow : UDINT;
  END_VAR

            VO_Event_Pulse := FALSE;
VO_Event_Code := 0;
VO_Event_Value := 0.0;

L_Alarm_Compat_All_OK := TRUE;
L_Alarm_First_Warning := '';
L_Alarm_First_Warning_Latched := FALSE;
L_Alarm_Shadow_Mismatch := FALSE;
L_Alarm_Shadow_First_Mismatch := 0;
L_Alarm_V2_Switch_Enabled := TRUE;
L_Alarm_V2_Path_Ready := FALSE;
L_Alarm_Using_Legacy_Fallback := TRUE;
L_Alarm_V2_Shadow_Compare_Enabled := TRUE;
L_Alarm_V2_Shadow_Diff_Found := FALSE;
L_Alarm_V2_Shadow_First_Diff_Slot := 0;
L_Alarm_V2_Event_Pulse := FALSE;
L_Alarm_V2_Event_Code := 0;
L_Alarm_V2_Event_Value := 0.0;
L_Alarm_V2_Next_ID_Shadow := VIO_Next_Alarm_ID;
L_History_V2_Shadow_Diff_Found := FALSE;
L_History_V2_Shadow_First_Diff_Slot := 0;
L_BlackBox_V2_Shadow_Diff_Found := FALSE;

// 1. Детекция новых тревог (антидребезг + передний фронт)
T_Debounce_Gas(IN := VI_Gas_Alarm, PT := T#100ms, VI_System_Time_MS := VI_System_Time_MS);
T_Debounce_Fire(IN := VI_Fire_Alarm, PT := T#100ms, VI_System_Time_MS := VI_System_Time_MS);
T_Debounce_Flood(IN := VI_Flood_Alarm, PT := T#500ms, VI_System_Time_MS := VI_System_Time_MS);
T_Debounce_Security(IN := VI_Security_Alarm, PT := T#100ms, VI_System_Time_MS := VI_System_Time_MS);

R_Trig_Gas(CLK := T_Debounce_Gas.Q);
R_Trig_Fire(CLK := T_Debounce_Fire.Q);
R_Trig_Flood(CLK := T_Debounce_Flood.Q);
R_Trig_Security(CLK := T_Debounce_Security.Q);
R_Trig_First_Fault(CLK := VI_First_Fault_Active);
FOR L_i := 1 TO GVL_CONSTANTS.C_MAX_BOILERS DO
    R_Trig_Boiler[L_i](CLK := VI_Boiler_Errors[L_i]);
END_FOR;

// 2. Добавление новых тревог в список (Кольцевой буфер)
L_Pending_Count := 0;
L_Event_Pulse_Latched := FALSE;

IF R_Trig_Gas.Q AND L_Pending_Count < 10 THEN
    L_Pending_Count := L_Pending_Count + 1;
    L_Pending_Alarms[L_Pending_Count].Timestamp_MS := VI_System_Time_MS;
    L_Pending_Alarms[L_Pending_Count].Source := 'Gas';
    L_Pending_Alarms[L_Pending_Count].Source_ID := 0;
    L_Pending_Alarms[L_Pending_Count].Message := 'Критическая концентрация газа!';
    L_Pending_Alarms[L_Pending_Count].Severity := E_ALERT_PRIORITY.ALERT_PRIORITY_CRITICAL;
    L_Pending_Alarms[L_Pending_Count].Is_Active := TRUE;
    L_Pending_Alarms[L_Pending_Count].Is_Acknowledged := FALSE;
END_IF;

IF R_Trig_Fire.Q AND L_Pending_Count < 10 THEN
    L_Pending_Count := L_Pending_Count + 1;
    L_Pending_Alarms[L_Pending_Count].Timestamp_MS := VI_System_Time_MS;
    L_Pending_Alarms[L_Pending_Count].Source := 'Fire';
    L_Pending_Alarms[L_Pending_Count].Source_ID := 0;
    L_Pending_Alarms[L_Pending_Count].Message := 'Обнаружено задымление!';
    L_Pending_Alarms[L_Pending_Count].Severity := E_ALERT_PRIORITY.ALERT_PRIORITY_CRITICAL;
    L_Pending_Alarms[L_Pending_Count].Is_Active := TRUE;
    L_Pending_Alarms[L_Pending_Count].Is_Acknowledged := FALSE;
END_IF;

IF R_Trig_Flood.Q AND L_Pending_Count < 10 THEN
    L_Pending_Count := L_Pending_Count + 1;
    L_Pending_Alarms[L_Pending_Count].Timestamp_MS := VI_System_Time_MS;
    L_Pending_Alarms[L_Pending_Count].Source := 'Flood';
    L_Pending_Alarms[L_Pending_Count].Source_ID := 0;
    L_Pending_Alarms[L_Pending_Count].Message := 'Обнаружена протечка воды!';
    L_Pending_Alarms[L_Pending_Count].Severity := E_ALERT_PRIORITY.ALERT_PRIORITY_CRITICAL;
    L_Pending_Alarms[L_Pending_Count].Is_Active := TRUE;
    L_Pending_Alarms[L_Pending_Count].Is_Acknowledged := FALSE;
END_IF;

IF R_Trig_Security.Q AND L_Pending_Count < 10 THEN
    L_Pending_Count := L_Pending_Count + 1;
    L_Pending_Alarms[L_Pending_Count].Timestamp_MS := VI_System_Time_MS;
    L_Pending_Alarms[L_Pending_Count].Source := 'Security';
    L_Pending_Alarms[L_Pending_Count].Source_ID := 0;
    L_Pending_Alarms[L_Pending_Count].Message := VI_Security_Msg;
    L_Pending_Alarms[L_Pending_Count].Severity := E_ALERT_PRIORITY.ALERT_PRIORITY_CRITICAL;
    L_Pending_Alarms[L_Pending_Count].Is_Active := TRUE;
    L_Pending_Alarms[L_Pending_Count].Is_Acknowledged := FALSE;
END_IF;

IF R_Trig_First_Fault.Q AND L_Pending_Count < 10 THEN
    L_Pending_Count := L_Pending_Count + 1;
    L_Pending_Alarms[L_Pending_Count].Timestamp_MS := VI_System_Time_MS;
    L_Pending_Alarms[L_Pending_Count].Source := 'Diagnostics';
    L_Pending_Alarms[L_Pending_Count].Source_ID := TO_BYTE(VI_First_Fault_Source);

    CASE VI_First_Fault_Type OF
        1: L_First_Fault_Type_Text := 'IO';
        2: L_First_Fault_Type_Text := 'Sensor';
        3: L_First_Fault_Type_Text := 'Comm';
        4: L_First_Fault_Type_Text := 'Subsystem';
        ELSE L_First_Fault_Type_Text := 'Unknown';
    END_CASE;

    CASE VI_First_Fault_Source OF
        1: L_First_Fault_Source_Text := 'Heating';
        2: L_First_Fault_Source_Text := 'DHW';
        3: L_First_Fault_Source_Text := 'Ventilation';
        4: L_First_Fault_Source_Text := 'Lighting';
        5: L_First_Fault_Source_Text := 'Access';
        ELSE L_First_Fault_Source_Text := 'Unknown';
    END_CASE;

    L_Pending_Alarms[L_Pending_Count].Message := CONCAT('Diagnostics root cause: ', CONCAT(L_First_Fault_Source_Text, CONCAT(' / ', L_First_Fault_Type_Text)));
    L_Pending_Alarms[L_Pending_Count].Severity := E_ALERT_PRIORITY.ALERT_PRIORITY_HIGH;
    L_Pending_Alarms[L_Pending_Count].Is_Active := TRUE;
    L_Pending_Alarms[L_Pending_Count].Is_Acknowledged := FALSE;
END_IF;

FOR L_j := 1 TO GVL_CONSTANTS.C_MAX_BOILERS DO
    IF R_Trig_Boiler[L_j].Q AND L_Pending_Count < 10 THEN
        L_Pending_Count := L_Pending_Count + 1;
        L_Pending_Alarms[L_Pending_Count].Timestamp_MS := VI_System_Time_MS;
        L_Pending_Alarms[L_Pending_Count].Source := 'Boiler';
        L_Pending_Alarms[L_Pending_Count].Source_ID := TO_BYTE(L_j);
        L_Pending_Alarms[L_Pending_Count].Message := CONCAT('Авария котла №', INT_TO_STRING(L_j));
        L_Pending_Alarms[L_Pending_Count].Severity := E_ALERT_PRIORITY.ALERT_PRIORITY_HIGH;
        L_Pending_Alarms[L_Pending_Count].Is_Active := TRUE;
        L_Pending_Alarms[L_Pending_Count].Is_Acknowledged := FALSE;
    END_IF;
END_FOR;

// Shadow comparison: execute Alarm V2 core on a separate shadow list.
// Legacy path remains authoritative; this is diagnostics only.
IF L_Alarm_V2_Shadow_Compare_Enabled THEN
    fbAlarmV2Core(
        VI_System_Time_MS := VI_System_Time_MS,
        VI_Pending_Alarms := L_Pending_Alarms,
        VIO_Alarm_List := L_Alarm_V2_List_Shadow,
        VIO_Next_Alarm_ID := L_Alarm_V2_Next_ID_Shadow,
        VO_Event_Pulse => L_Alarm_V2_Event_Pulse,
        VO_Event_Code => L_Alarm_V2_Event_Code,
        VO_Event_Value => L_Alarm_V2_Event_Value
    );
END_IF;

// Staging integration: Alarm V2 core is called behind the phase-4 switch scaffold.
// Current state: switch remains disabled, so legacy path stays authoritative.
IF L_Alarm_V2_Switch_Enabled AND L_Alarm_V2_Path_Ready THEN
    fbAlarmV2Core(
        VI_System_Time_MS := VI_System_Time_MS,
        VI_Pending_Alarms := L_Pending_Alarms,
        VIO_Alarm_List := VO_Alarm_List,
        VIO_Next_Alarm_ID := VIO_Next_Alarm_ID
    );
END_IF;

// Обработка очереди новых тревог с учетом приоритетов
FOR L_i := 1 TO L_Pending_Count DO
    fbCompatAlarm[L_i](VI_Alarm_Legacy := L_Pending_Alarms[L_i]);

    IF NOT fbCompatAlarm[L_i].VO_OK THEN
        L_Alarm_Compat_All_OK := FALSE;
    END_IF;

    IF (NOT L_Alarm_First_Warning_Latched) AND (NOT fbCompatAlarm[L_i].VO_OK) THEN
        L_Alarm_First_Warning := 'Translation issue';
        L_Alarm_First_Warning_Latched := TRUE;
    END_IF;

    IF fbCompatAlarm[L_i].VO_Alarm_Legacy_Roundtrip.ID <> L_Pending_Alarms[L_i].ID THEN
        L_Alarm_Shadow_Mismatch := TRUE;
        IF L_Alarm_Shadow_First_Mismatch = 0 THEN
            L_Alarm_Shadow_First_Mismatch := L_i;
        END_IF;
    END_IF;
    // Phase 4 scaffold: optional Alarm V2 switch point.
    // Current state: always remain on legacy behavior.
    // Future state: when Alarm V2 path is implemented and validated,
    // this block becomes the controlled branch point.
    IF L_Alarm_V2_Switch_Enabled AND L_Alarm_V2_Path_Ready THEN
        L_Alarm_Using_Legacy_Fallback := FALSE;
        // Guarded V2 pipeline is allowed by shadow validation.
        // Current runtime logic still keeps legacy action flow authoritative until next package.
    ELSE
        L_Alarm_Using_Legacy_Fallback := TRUE;
    END_IF;

    L_Target_Slot := 0;
    
    // 1. Ищем пустой слот
    FOR L_k := 1 TO GVL_CONSTANTS.C_MAX_ALARMS DO
        IF VO_Alarm_List[L_k].ID = 0 THEN
            L_Target_Slot := L_k;
            EXIT;
        END_IF;
    END_FOR;
    
    // 2. Ищем квитированную тревогу с наименьшим приоритетом
    IF L_Target_Slot = 0 THEN
        L_Min_Pri := 999;
        FOR L_k := 1 TO GVL_CONSTANTS.C_MAX_ALARMS DO
            IF VO_Alarm_List[L_k].Is_Acknowledged AND TO_INT(VO_Alarm_List[L_k].Severity) < L_Min_Pri THEN
                L_Min_Pri := TO_INT(VO_Alarm_List[L_k].Severity);
                L_Target_Slot := L_k;
            END_IF;
        END_FOR;
    END_IF;
    
    // 3. Ищем неквитированную тревогу с наименьшим приоритетом (если он ниже добавляемой)
    IF L_Target_Slot = 0 THEN
        L_Min_Pri := 999;
        FOR L_k := 1 TO GVL_CONSTANTS.C_MAX_ALARMS DO
            IF TO_INT(VO_Alarm_List[L_k].Severity) < L_Min_Pri AND TO_INT(VO_Alarm_List[L_k].Severity) < TO_INT(L_Pending_Alarms[L_i].Severity) THEN
                L_Min_Pri := TO_INT(VO_Alarm_List[L_k].Severity);
                L_Target_Slot := L_k;
            END_IF;
        END_FOR;
    END_IF;
    
    IF L_Target_Slot = 0 THEN 
        // Буфер полон критических неквитированных тревог. Не затираем!
        CONTINUE; 
    END_IF;
    
    VO_Alarm_List[L_Target_Slot] := L_Pending_Alarms[L_i];
    VO_Alarm_List[L_Target_Slot].ID := VIO_Next_Alarm_ID;
    VIO_Next_Alarm_ID := VIO_Next_Alarm_ID + 1;
    IF VIO_Next_Alarm_ID = 0 THEN VIO_Next_Alarm_ID := 1; END_IF;
    IF NOT L_Event_Pulse_Latched THEN
        VO_Event_Pulse := TRUE;
        VO_Event_Code := 1203;
        VO_Event_Value := TO_REAL(VO_Alarm_List[L_Target_Slot].Severity);
        L_Event_Pulse_Latched := TRUE;
    END_IF;
END_FOR;

// Shadow comparison results: compare legacy output and V2 shadow output.
IF L_Alarm_V2_Shadow_Compare_Enabled THEN
    FOR L_i := 1 TO GVL_CONSTANTS.C_MAX_ALARMS DO
        IF (VO_Alarm_List[L_i].ID <> L_Alarm_V2_List_Shadow[L_i].ID)
           OR (VO_Alarm_List[L_i].Is_Active <> L_Alarm_V2_List_Shadow[L_i].Is_Active)
           OR (VO_Alarm_List[L_i].Is_Acknowledged <> L_Alarm_V2_List_Shadow[L_i].Is_Acknowledged)
           OR (VO_Alarm_List[L_i].Severity <> L_Alarm_V2_List_Shadow[L_i].Severity) THEN
            L_Alarm_V2_Shadow_Diff_Found := TRUE;
            IF L_Alarm_V2_Shadow_First_Diff_Slot = 0 THEN
                L_Alarm_V2_Shadow_First_Diff_Slot := L_i;
            END_IF;
        END_IF;
    END_FOR;
END_IF;

// 3. Обновление статуса существующих тревог (ушли ли они?)
FOR L_i := 1 TO GVL_CONSTANTS.C_MAX_ALARMS DO
    IF VO_Alarm_List[L_i].ID <> 0 THEN
        IF VO_Alarm_List[L_i].Source = 'Gas' THEN VO_Alarm_List[L_i].Is_Active := VI_Gas_Alarm;
        ELSIF VO_Alarm_List[L_i].Source = 'Fire' THEN VO_Alarm_List[L_i].Is_Active := VI_Fire_Alarm;
        ELSIF VO_Alarm_List[L_i].Source = 'Flood' THEN VO_Alarm_List[L_i].Is_Active := VI_Flood_Alarm;
        ELSIF VO_Alarm_List[L_i].Source = 'Security' THEN VO_Alarm_List[L_i].Is_Active := VI_Security_Alarm;
        ELSIF VO_Alarm_List[L_i].Source = 'Diagnostics' THEN VO_Alarm_List[L_i].Is_Active := VI_First_Fault_Active;
        ELSIF VO_Alarm_List[L_i].Source = 'Boiler' THEN 
            IF TO_INT(VO_Alarm_List[L_i].Source_ID) >= 1 AND TO_INT(VO_Alarm_List[L_i].Source_ID) <= GVL_CONSTANTS.C_MAX_BOILERS THEN
                VO_Alarm_List[L_i].Is_Active := VI_Boiler_Errors[TO_INT(VO_Alarm_List[L_i].Source_ID)];
            END_IF;
        END_IF;
    END_IF;
END_FOR;

// 4. Квитирование тревог
IF VI_Acknowledge_All THEN
    FOR L_i := 1 TO GVL_CONSTANTS.C_MAX_ALARMS DO
        IF VO_Alarm_List[L_i].ID <> 0 THEN
            VO_Alarm_List[L_i].Is_Acknowledged := TRUE;
        END_IF;
    END_FOR;

    IF NOT L_Event_Pulse_Latched THEN
        VO_Event_Pulse := TRUE;
        VO_Event_Code := 1201;
        VO_Event_Value := TO_REAL(VO_Unacked_Count);
        L_Event_Pulse_Latched := TRUE;
    END_IF;
END_IF;

// 4.5 Автоквитирование некритичных тревог, если они больше не активны
FOR L_i := 1 TO GVL_CONSTANTS.C_MAX_ALARMS DO
    IF VO_Alarm_List[L_i].ID <> 0 AND NOT VO_Alarm_List[L_i].Is_Active AND NOT VO_Alarm_List[L_i].Is_Acknowledged THEN
        IF VO_Alarm_List[L_i].Severity <> E_ALERT_PRIORITY.ALERT_PRIORITY_CRITICAL THEN
            VO_Alarm_List[L_i].Is_Acknowledged := TRUE;
        END_IF;
    END_IF;
END_FOR;

// 5. Очистка списка (удаление неактивных И квитированных тревог)
// В кольцевом буфере мы просто помечаем слот как пустой (ID = 0), без сдвига массива
FOR L_i := 1 TO GVL_CONSTANTS.C_MAX_ALARMS DO
    IF VO_Alarm_List[L_i].ID <> 0 AND NOT VO_Alarm_List[L_i].Is_Active AND VO_Alarm_List[L_i].Is_Acknowledged THEN
        // Удаляем тревогу
        VO_Alarm_List[L_i].ID := 0;
        IF NOT L_Event_Pulse_Latched THEN
            VO_Event_Pulse := TRUE;
            VO_Event_Code := 1202;
            VO_Event_Value := 0.0;
            L_Event_Pulse_Latched := TRUE;
        END_IF;
    END_IF;
END_FOR;

// Shadow bridge: Alarm -> History V2 (diagnostic only)
fbHistoryV2Core(
    VI_Event_Pulse := VO_Event_Pulse,
    VI_Event_Code := VO_Event_Code,
    VI_Event_Value := VO_Event_Value,
    VI_System_Time_MS := VI_System_Time_MS,
    VIO_History_Buffer := L_History_V2_Buffer_Shadow
);

// Shadow bridge: System -> BlackBox V2 (diagnostic only)
fbBlackBoxV2Core(
    VI_System_Time_MS := VI_System_Time_MS,
    VI_System_Mode := 0,
    VI_Critical_Alarm_Active := VO_Global_Critical,
    VI_Warning_Active := VO_Global_Warning,
    VI_First_Fault_Type := TO_BYTE(VI_First_Fault_Type),
    VI_First_Fault_Source := TO_BYTE(VI_First_Fault_Source),
    VI_Gas_Alarm := VI_Gas_Alarm,
    VI_Fire_Alarm := VI_Fire_Alarm,
    VI_Flood_Alarm := VI_Flood_Alarm,
    VO_Snapshot => L_BlackBox_V2_Snapshot_Shadow
);

// Shadow validation: History V2 / BlackBox V2
IF VO_Event_Pulse THEN
    IF (L_History_V2_Buffer_Shadow[1].Event_Code <> VO_Event_Code)
       OR (ABS(L_History_V2_Buffer_Shadow[1].Event_Value - VO_Event_Value) > 0.0001) THEN
        L_History_V2_Shadow_Diff_Found := TRUE;
        IF L_History_V2_Shadow_First_Diff_Slot = 0 THEN
            L_History_V2_Shadow_First_Diff_Slot := 1;
        END_IF;
    END_IF;
END_IF;

IF (L_BlackBox_V2_Snapshot_Shadow.Gas_Alarm <> VI_Gas_Alarm)
   OR (L_BlackBox_V2_Snapshot_Shadow.Fire_Alarm <> VI_Fire_Alarm)
   OR (L_BlackBox_V2_Snapshot_Shadow.Flood_Alarm <> VI_Flood_Alarm)
   OR (L_BlackBox_V2_Snapshot_Shadow.First_Fault_Type <> TO_BYTE(VI_First_Fault_Type))
   OR (L_BlackBox_V2_Snapshot_Shadow.First_Fault_Source <> TO_BYTE(VI_First_Fault_Source)) THEN
    L_BlackBox_V2_Shadow_Diff_Found := TRUE;
END_IF;

// Guarded V2 pipeline enable:
// V2 path is allowed only when no shadow diff is present in Alarm/History/BlackBox.
IF L_Alarm_V2_Switch_Enabled THEN
    IF (NOT L_Alarm_V2_Shadow_Diff_Found)
       AND (NOT L_History_V2_Shadow_Diff_Found)
       AND (NOT L_BlackBox_V2_Shadow_Diff_Found) THEN
        L_Alarm_V2_Path_Ready := TRUE;
        L_Alarm_Using_Legacy_Fallback := FALSE;
    ELSE
        L_Alarm_V2_Path_Ready := FALSE;
        L_Alarm_Using_Legacy_Fallback := TRUE;
    END_IF;
ELSE
    L_Alarm_V2_Path_Ready := FALSE;
    L_Alarm_Using_Legacy_Fallback := TRUE;
END_IF;

// 6. Подсчет статистики и формирование глобальных флагов
VO_Global_Critical := FALSE;
VO_Global_Warning := FALSE;
VO_Siren_Active := FALSE;
VO_Active_Count := 0;
VO_Unacked_Count := 0;

FOR L_i := 1 TO GVL_CONSTANTS.C_MAX_ALARMS DO
    IF VO_Alarm_List[L_i].ID <> 0 THEN
        IF VO_Alarm_List[L_i].Is_Active THEN
            VO_Active_Count := VO_Active_Count + 1;
        END_IF;
        
        IF NOT VO_Alarm_List[L_i].Is_Acknowledged THEN
            VO_Unacked_Count := VO_Unacked_Count + 1;
            
            IF VO_Alarm_List[L_i].Severity = E_ALERT_PRIORITY.ALERT_PRIORITY_CRITICAL THEN
                VO_Global_Critical := TRUE;
                // Сирена работает только для неквитированных критических тревог, если не включен Mute
                IF NOT VI_Mute_Siren THEN
                    VO_Siren_Active := TRUE;
                END_IF;
            ELSIF VO_Alarm_List[L_i].Severity = E_ALERT_PRIORITY.ALERT_PRIORITY_HIGH THEN
                VO_Global_Warning := TRUE;
            END_IF;
        END_IF;
    END_IF;
END_FOR;
// >>> BULK_SYNC_ANCHOR: FB_Alarm_Manager <<<
          
END_FUNCTION_BLOCK

FUNCTION_BLOCK FB_Sensor_Analog_Processing
  VAR_INPUT
    VI_Raw_Value : WORD;
    VI_Sensor_Type : INT := 0;
    VI_Min_Scale : REAL;
    VI_Max_Scale : REAL;
    VI_Offset : REAL;
    VI_Multiplier : REAL := 1.0;
    VI_Filter_Time_MS : UDINT := GVL_CONSTANTS.C_MS_IN_SECOND;
    VI_System_Time_MS : UDINT;
    VI_Fallback_Mode : INT := 0;
    VI_Default_Value : REAL := 0.0;
  END_VAR
  VAR_OUTPUT
    VO_Value : REAL;
    VO_Error : BOOL;
    VO_Diag_Code : WORD;
  END_VAR
  VAR
    L_Scaled : REAL;
    L_Filtered : REAL;
    L_History : ARRAY[0..9] OF REAL;
    L_History_Idx : INT := 0;
    L_History_Sum : REAL := 0.0;
    L_History_Count : INT := 0;
    L_Last_Time : UDINT;
    L_DT : UDINT;
    L_First_Scan : BOOL := TRUE;
    L_i : INT;
  END_VAR

            // 1. Error checking and scaling based on sensor type
VO_Error := FALSE;
VO_Diag_Code := 0;

CASE VI_Sensor_Type OF
    0: // 4-20mA (NAMUR NE43: < 3.6mA or > 21mA)
        IF VI_Raw_Value < GVL_CONSTANTS.C_ANALOG_3_6MA_RAW THEN // < 3.6mA (Open circuit)
            VO_Error := TRUE;
            VO_Diag_Code := 1;
        ELSIF VI_Raw_Value > GVL_CONSTANTS.C_ANALOG_21MA_RAW THEN // > 21mA (Short circuit)
            VO_Error := TRUE;
            VO_Diag_Code := 2;
        ELSE
            // 4mA = 5529, 20mA = 27648
            L_Scaled := VI_Min_Scale + (TO_REAL(VI_Raw_Value - GVL_CONSTANTS.C_ANALOG_4MA_RAW) / TO_REAL(GVL_CONSTANTS.C_ANALOG_RAW_MAX - GVL_CONSTANTS.C_ANALOG_4MA_RAW)) * (VI_Max_Scale - VI_Min_Scale);
        END_IF;
        
    1: // 0-10V (0-27648)
        IF VI_Raw_Value > GVL_CONSTANTS.C_ANALOG_10V_MAX_RAW THEN // Out of range
            VO_Error := TRUE;
            VO_Diag_Code := 3;
        ELSE
            L_Scaled := VI_Min_Scale + (TO_REAL(VI_Raw_Value) / TO_REAL(GVL_CONSTANTS.C_ANALOG_RAW_MAX)) * (VI_Max_Scale - VI_Min_Scale);
        END_IF;
        
    2: // PT100/1000 (Direct temperature * 10, e.g., 255 = 25.5C)
        // Typically, 16-bit signed integer for temperature
        IF VI_Raw_Value = 16#7FFF OR VI_Raw_Value = 16#8000 THEN // Sensor error codes
            VO_Error := TRUE;
            VO_Diag_Code := 1;
        ELSE
            L_Scaled := TO_REAL(TO_INT(VI_Raw_Value)) / 10.0;
            IF L_Scaled < VI_Min_Scale OR L_Scaled > VI_Max_Scale THEN
                VO_Error := TRUE;
                VO_Diag_Code := 3;
            END_IF;
        END_IF;
        
    ELSE
        VO_Error := TRUE;
        VO_Diag_Code := 16#FFFF; // Unknown sensor type
END_CASE;

// 2. Fallback handling
IF VO_Error THEN
    IF VI_Fallback_Mode = 1 THEN
        VO_Value := VI_Default_Value;
    END_IF;
    // If VI_Fallback_Mode = 0, VO_Value retains its last good value (L_Filtered)
    RETURN;
END_IF;

// 3. Calibration
L_Scaled := (L_Scaled * VI_Multiplier) + VI_Offset;

// 4. Moving Average Filter (ТЗ 1.2)
IF L_First_Scan THEN
    L_Filtered := L_Scaled;
    L_First_Scan := FALSE;
    L_Last_Time := VI_System_Time_MS;
    
    // Инициализация массива истории
    FOR L_i := 0 TO 9 DO
        L_History[L_i] := L_Scaled;
    END_FOR;
    L_History_Sum := L_Scaled * 10.0;
    L_History_Count := 10;
    L_History_Idx := 0;
END_IF;

L_DT := (SEL(VI_System_Time_MS >= L_Last_Time, VI_System_Time_MS - L_Last_Time, (4294967295 - L_Last_Time) + VI_System_Time_MS + 1));
IF VI_Filter_Time_MS = 0 THEN
    L_Filtered := L_Scaled;
    L_Last_Time := VI_System_Time_MS;
ELSIF L_DT >= (VI_Filter_Time_MS / 10) THEN // Обновляем 10 раз за время фильтрации
    // Вычитаем старое значение
    L_History_Sum := L_History_Sum - L_History[L_History_Idx];
    
    // Добавляем новое значение
    L_History[L_History_Idx] := L_Scaled;
    L_History_Sum := L_History_Sum + L_Scaled;
    
    // Сдвигаем индекс
    L_History_Idx := (L_History_Idx + 1) MOD 10;
    
    // Вычисляем среднее
    L_Filtered := L_History_Sum / 10.0;
    
    L_Last_Time := VI_System_Time_MS;
END_IF;

VO_Value := L_Filtered;
          
END_FUNCTION_BLOCK

FUNCTION_BLOCK FB_History_V2_Core
  VAR_INPUT
    VI_Event_Pulse : BOOL;
    VI_Event_Code : UDINT;
    VI_Event_Value : REAL;
    VI_System_Time_MS : UDINT;
  END_VAR
  VAR_IN_OUT
    VIO_History_Buffer : ARRAY[1..GVL_CONSTANTS.C_MAX_HISTORY_RECORDS] OF ST_History_Event_V2;
  END_VAR

            IF VI_Event_Pulse THEN
    VIO_History_Buffer[1].Event_Code := TO_UINT(VI_Event_Code);
    VIO_History_Buffer[1].Event_Value := VI_Event_Value;
END_IF;
          
END_FUNCTION_BLOCK

FUNCTION_BLOCK FB_Sensor_Calibration
  VAR_INPUT
    VI_Sensor_ID : UDINT;
    VI_Reference_Value : REAL;
    VI_Current_Value : REAL;
    VI_Apply : BOOL;
  END_VAR
  VAR_OUTPUT
    VO_Offset : REAL;
    VO_Multiplier : REAL := 1.0;
    VO_Done : BOOL;
  END_VAR
  VAR
    L_Applied : BOOL;
  END_VAR

            IF VI_Apply AND NOT L_Applied THEN
    // Простая калибровка смещением (одноточечная)
    VO_Offset := VI_Reference_Value - VI_Current_Value;
    VO_Done := TRUE;
    L_Applied := TRUE;
ELSIF NOT VI_Apply THEN
    VO_Done := FALSE;
    L_Applied := FALSE;
END_IF;
          
END_FUNCTION_BLOCK

FUNCTION_BLOCK FB_Scenario_Manager
  VAR_INPUT
    VI_System_Time_MS : UDINT;
    VI_Activate_Request : E_SCENARIO_TYPE;
    VI_IsActivePLC : BOOL;
    VI_System_Mode : E_System_Operating_Mode;
  END_VAR
  VAR_OUTPUT
    VO_Current_Scenario : E_SCENARIO_TYPE;
    VO_Status_Msg : STRING(200);
  END_VAR
  VAR
    L_Last_Scenario_Time : UDINT;
  END_VAR

            IF NOT VI_IsActivePLC THEN
    RETURN;
END_IF;

CASE VI_System_Mode OF
    E_System_Operating_Mode.MODE_SAFE_STOP,
    E_System_Operating_Mode.MODE_FREEZE_PROTECTION:
        IF VO_Current_Scenario <> E_SCENARIO_TYPE.SCENARIO_NONE THEN
            VO_Current_Scenario := E_SCENARIO_TYPE.SCENARIO_NONE;
            VO_Status_Msg := 'Сценарии принудительно отключены режимом безопасности';
        END_IF;
        RETURN;

    E_System_Operating_Mode.MODE_DEGRADED:
        VO_Status_Msg := 'Смена сценариев заблокирована: деградированный режим';
        RETURN;
END_CASE;

IF VI_Activate_Request <> VO_Current_Scenario THEN
    // Проверка минимального времени работы сценария
    IF (VI_System_Time_MS - L_Last_Scenario_Time) >= 60000 OR VO_Current_Scenario = E_SCENARIO_TYPE.SCENARIO_NONE THEN
        // Логика переключения сценариев
        VO_Current_Scenario := VI_Activate_Request;
        L_Last_Scenario_Time := VI_System_Time_MS;
        
        CASE VO_Current_Scenario OF
        E_SCENARIO_TYPE.SCENARIO_NONE:
            VO_Status_Msg := 'Сценарии отключены';
        E_SCENARIO_TYPE.SCENARIO_AWAY:
            VO_Status_Msg := 'Активирован сценарий: Вне дома (Охрана + Энергосбережение)';
        E_SCENARIO_TYPE.SCENARIO_SLEEP:
            VO_Status_Msg := 'Активирован сценарий: Сон (Ночное освещение + Климат)';
        E_SCENARIO_TYPE.SCENARIO_PRESENCE:
            VO_Status_Msg := 'Активирован сценарий: Имитация присутствия';
        END_CASE;
    END_IF;
END_IF;
// >>> BULK_SYNC_ANCHOR: FB_Scenario_Manager <<<
          
END_FUNCTION_BLOCK

FUNCTION_BLOCK FB_Gas_Valve_Controller
  VAR_INPUT
    VI_System_Time : UDINT;
    VI_IsActivePLC : BOOL;
    VI_Gas_Alarm : BOOL;
    VI_Config : ST_Gas_Valve_Configuration;
  END_VAR
  VAR_INPUT
    VI_Operator_ID : STRING(10);
    VI_Force : BOOL;
  END_VAR
  VAR_INPUT
    VI_Operator_ID : STRING(10);
    VI_Force : BOOL;
  END_VAR
  VAR_OUTPUT
    VO_Valve_Closed : BOOL;
    VO_Status_Msg : STRING(200);
  END_VAR

            // При аварии газа - немедленное закрытие
IF VI_Gas_Alarm AND VI_IsActivePLC THEN
    VO_Valve_Closed := TRUE;
    VO_Status_Msg := 'ГАЗОВЫЙ КЛАПАН ЗАКРЫТ ПО АВАРИИ';
END_IF;
          

METHOD OpenValve : BOOL
                  IF VI_IsActivePLC OR VI_Force THEN
    VO_Valve_Closed := FALSE;
    OpenValve := TRUE;
END_IF;
                
END_METHOD

METHOD CloseValve : BOOL
                  VO_Valve_Closed := TRUE;
CloseValve := TRUE;
                
END_METHOD

METHOD GetStatus : BYTE
                  GetStatus := TO_BYTE(SEL(VO_Valve_Closed, 0, 1));
                
END_METHOD
END_FUNCTION_BLOCK

FUNCTION_BLOCK FB_State_Manager
  VAR_INPUT
    VI_System_Severity : E_System_Severity;
    VI_Root_Cause : E_System_Root_Cause;
    VI_Freeze_Risk : BOOL := FALSE;
  END_VAR
  VAR_OUTPUT
    VO_System_OK : BOOL;
    VO_System_Warning : BOOL;
    VO_System_Critical : BOOL;
    VO_Status_Msg : STRING(200);
    VO_System_Mode : E_System_Operating_Mode;
  END_VAR

            VO_System_OK := FALSE;
VO_System_Warning := FALSE;
VO_System_Critical := FALSE;
VO_Status_Msg := '';
VO_System_Mode := E_System_Operating_Mode.MODE_NORMAL;

CASE VI_System_Severity OF
    E_System_Severity.SEV_NORMAL:
        VO_System_OK := TRUE;
        VO_Status_Msg := 'Система в норме';
        VO_System_Mode := E_System_Operating_Mode.MODE_NORMAL;

    E_System_Severity.SEV_WARNING:
        VO_System_Warning := TRUE;
        VO_System_Mode := E_System_Operating_Mode.MODE_DEGRADED;
        CASE VI_Root_Cause OF
            E_System_Root_Cause.ROOT_WATER_LEAK:
                VO_Status_Msg := 'Предупреждение: протечка воды';
            E_System_Root_Cause.ROOT_CO_WARNING:
                VO_Status_Msg := 'Предупреждение: повышенный CO';
            ELSE
                VO_Status_Msg := 'Предупреждение системы';
        END_CASE;

